Omron Sysmac Studio project Meca500_V9_1_5_Omron_EtherCat_Square_Demo_V1 (Sysmac Studio 1.47.0.64008, StandardProject)

# Controller NX1P2_9024DT1: NX1P2-9024DT1 version 1.16
Units and slaves: Node1 : Meca500 (E001)
Task PrimaryTask (priority 4, period or condition 2000): Meca500_IOs, Meca500_Sequence, Meca500_Instructions

TYPE RobotControl : STRUCT
    Deactivate : BOOL;  (* offset 0.0 *)
    Activate : BOOL;  (* offset 0.1 *)
    Home : BOOL;  (* offset 0.2 *)
    ResetError : BOOL;  (* offset 0.3 *)
    EnableSimulation : BOOL;  (* offset 0.4 *)
    EnableRecoveryMode : BOOL;  (* offset 0.5 *)
END_STRUCT END_TYPE
TYPE Meca500 : STRUCT
    Outputs : Outputs;
    Inputs : Inputs;
    CommandsID : Meca500Cmd;
END_STRUCT END_TYPE
TYPE Inputs : STRUCT
    Status : Status;  (* offset 0.0 *)
    Motion : Motion;  (* offset 4.0 *)
    Joint_Set : Joint_Set;  (* offset 16.0 *)
    EndEffector_Pose : EndEffector_Pose;  (* offset 40.0 *)
    Configurations : Configurations;  (* offset 64.0 *)
    WRF : WRF;  (* offset 68.0 *)
    TRF : TRF;  (* offset 92.0 *)
    TimeStamp : TimeStamp;  (* offset 116.0 *)
    Reserved1 : SINT;  (* offset 128.0 *)
    Reserved2 : SINT;  (* offset 132.0 *)
    Reserved3 : SINT;  (* offset 136.0 *)
    DynamicData0 : DynamicData;  (* offset 140.0 *)
    DynamicData1 : DynamicData;  (* offset 168.0 *)
    DynamicData2 : DynamicData;  (* offset 196.0 *)
    DynamicData3 : DynamicData;  (* offset 224.0 *)
END_STRUCT END_TYPE
TYPE Status : STRUCT
    Busy : BOOL;
    Activated : BOOL;
    Homed : BOOL;
    SimActivated : BOOL;
    BrakesEngaged : BOOL;
    RecoveryMode : BOOL;
    Error : UINT;
END_STRUCT END_TYPE
TYPE Motion : STRUCT
    CheckPoint : UDINT;  (* offset 0.0 *)
    MoveID : UINT;  (* offset 4.0 *)
    FifoSpace : UINT;  (* offset 6.0 *)
    Paused : BOOL;  (* offset 8.0 *)
    EOB : BOOL;  (* offset 8.1 *)
    EOM : BOOL;  (* offset 8.2 *)
    FifoCleared : BOOL;  (* offset 8.3 *)
    PStop : BOOL;  (* offset 8.4 *)
    ExcessiveTorque : BOOL;  (* offset 8.5 *)
    OfflineProgramID : UINT;  (* offset 10.0 *)
END_STRUCT END_TYPE
TYPE Joint_Set : STRUCT
    SubIndex001 : REAL;
    SubIndex002 : REAL;
    SubIndex003 : REAL;
    SubIndex004 : REAL;
    SubIndex005 : REAL;
    SubIndex006 : REAL;
END_STRUCT END_TYPE
TYPE EndEffector_Pose : STRUCT
    SubIndex001 : REAL;
    SubIndex002 : REAL;
    SubIndex003 : REAL;
    SubIndex004 : REAL;
    SubIndex005 : REAL;
    SubIndex006 : REAL;
END_STRUCT END_TYPE
TYPE Configurations : STRUCT
    Shoulder : SINT;  (* offset 0.0 *)
    Elbow : SINT;  (* offset 1.0 *)
    Wrist : SINT;  (* offset 2.0 *)
    Turn : SINT;  (* offset 3.0 *)
END_STRUCT END_TYPE
TYPE WRF : STRUCT
    SubIndex001 : REAL;
    SubIndex002 : REAL;
    SubIndex003 : REAL;
    SubIndex004 : REAL;
    SubIndex005 : REAL;
    SubIndex006 : REAL;
END_STRUCT END_TYPE
TYPE TRF : STRUCT
    SubIndex001 : REAL;
    SubIndex002 : REAL;
    SubIndex003 : REAL;
    SubIndex004 : REAL;
    SubIndex005 : REAL;
    SubIndex006 : REAL;
END_STRUCT END_TYPE
TYPE TimeStamp : STRUCT
    Seconds : UDINT;
    MicroSeconds : UDINT;
    DynamicDataCycles : UDINT;
END_STRUCT END_TYPE
TYPE DynamicData : STRUCT
    DynamicDataType : UDINT;
    DynamicDataValue0 : REAL;
    DynamicDataValue1 : REAL;
    DynamicDataValue2 : REAL;
    DynamicDataValue3 : REAL;
    DynamicDataValue4 : REAL;
    DynamicDataValue5 : REAL;
END_STRUCT END_TYPE
TYPE Outputs : STRUCT
    RobotControl : RobotControl;  (* offset 0.0 *)
    MotionControl : MotionControl;  (* offset 4.0 *)
    MotionCommand : MotionCommand;  (* offset 8.0 *)
    HostTime : UDINT;  (* offset 36.0 *)
    BrakesControlAllowed : BOOL;  (* offset 40.0 *)
    BrakesEngaged : BOOL;  (* offset 40.1 *)
    DynamicDataCfg0 : UDINT;  (* offset 42.0 *)
    DynamicDataCfg1 : UDINT;  (* offset 46.0 *)
    DynamicDataCfg2 : UDINT;  (* offset 50.0 *)
    DynamicDataCfg3 : UDINT;  (* offset 56.0 *)
END_STRUCT END_TYPE
TYPE MotionControl : STRUCT
    MoveID : UINT;  (* offset 0.0 *)
    Setpoint : BOOL;  (* offset 2.0 *)
    Pause : BOOL;  (* offset 2.1 *)
    CleaMove : BOOL;  (* offset 2.2 *)
    ResetPStop2 : BOOL;  (* offset 2.3 *)
END_STRUCT END_TYPE
TYPE MotionCommand : STRUCT
    MoveCommand : UDINT;  (* offset 0.0 *)
    MoveSubIndex001 : REAL;  (* offset 4.0 *)
    MoveSubIndex002 : REAL;  (* offset 8.0 *)
    MoveSubIndex003 : REAL;  (* offset 12.0 *)
    MoveSubIndex004 : REAL;  (* offset 16.0 *)
    MoveSubIndex005 : REAL;  (* offset 20.0 *)
    MoveSubIndex006 : REAL;  (* offset 24.0 *)
END_STRUCT END_TYPE
TYPE Meca500Cmd : (NoCmd := 0, MoveJoints := 1, MovePose := 2, MoveLin := 3, MoveLinRelTrf := 4, MoveLinRelWrf := 5, Delay := 6, SetBlending := 7, SetJointVel := 8, SetJointAcc := 9, SetCartAngVel := 10, SetCartLinVel := 11, SetCartAcc := 12, SetTrf := 13, SetWrf := 14, SetConf := 15, SetAutoConf := 16, SetCheckpoint := 17, Gripper := 18, SetGripperVel := 19, SetGripperForce := 20, MoveJointsVel := 21, MoveLinVelWrf := 22, MoveLinVelTrf := 23, SetVelTimeout := 24, SetConfTurn := 25, SetAutoConfTurn := 26, SetTorqueLimits := 27, SetTorquesLimitCfg := 28, MoveJointsRel := 29, SetValveState := 30, SetGripperRange := 31, MoveGripper := 32, StartProgram := 100); END_TYPE

VAR_GLOBAL
    E001 : Meca500;  (* Robot Structure *)
    Position : ARRAY[0..5] OF real;  (* Array for positions *)
    StepSquareMove : INT;  (* Sequencer step *)
    MoveJoint1Buffered : BOOL;
    MovePose1Buffered : BOOL;
    MoveLin1Buffered : BOOL;
    SetCartLinVel1Buffered : BOOL;
    E001_Robot_Control_Deactivate_7200_01 : BOOL;  (* at ECAT://node#1/Robot Control_Deactivate_7200_01 *)
    E001_Robot_Control_Activate_7200_02 : BOOL;  (* at ECAT://node#1/Robot Control_Activate_7200_02 *)
    E001_Robot_Control_Home_7200_03 : BOOL;  (* at ECAT://node#1/Robot Control_Home_7200_03 *)
    E001_Robot_Control_Reset_Error_7200_04 : BOOL;  (* at ECAT://node#1/Robot Control_Reset Error_7200_04 *)
    E001_Robot_Control_Sim_Mode_7200_05 : BOOL;  (* at ECAT://node#1/Robot Control_Sim Mode_7200_05 *)
    E001_Robot_Control_Recovery_Mode_7200_06 : BOOL;  (* at ECAT://node#1/Robot Control_Recovery Mode_7200_06 *)
    E001_Motion_Control_Move_ID_7310_01 : UINT;  (* at ECAT://node#1/Motion Control_Move ID_7310_01 *)
    E001_Motion_Control_SetPoint_7310_02 : BOOL;  (* at ECAT://node#1/Motion Control_SetPoint_7310_02 *)
    E001_Motion_Control_Pause_7310_03 : BOOL;  (* at ECAT://node#1/Motion Control_Pause_7310_03 *)
    E001_Motion_Control_Clear_Move_7310_04 : BOOL;  (* at ECAT://node#1/Motion Control_Clear Move_7310_04 *)
    E001_Motion_Control_Reset_PStop2_7310_05 : BOOL;  (* at ECAT://node#1/Motion Control_Reset PStop2_7310_05 *)
    E001_Move_Move_Command_7305_00 : UDINT;  (* at ECAT://node#1/Move_Move Command_7305_00 *)
    E001_Move_SubIndex_001_7306_01 : REAL;  (* at ECAT://node#1/Move_SubIndex 001_7306_01 *)
    E001_Move_SubIndex_002_7306_02 : REAL;  (* at ECAT://node#1/Move_SubIndex 002_7306_02 *)
    E001_Move_SubIndex_003_7306_03 : REAL;  (* at ECAT://node#1/Move_SubIndex 003_7306_03 *)
    E001_Move_SubIndex_004_7306_04 : REAL;  (* at ECAT://node#1/Move_SubIndex 004_7306_04 *)
    E001_Move_SubIndex_005_7306_05 : REAL;  (* at ECAT://node#1/Move_SubIndex 005_7306_05 *)
    E001_Move_SubIndex_006_7306_06 : REAL;  (* at ECAT://node#1/Move_SubIndex 006_7306_06 *)
    E001_Host_Time_Host_Time_7400_00 : UDINT;  (* at ECAT://node#1/Host Time_Host Time_7400_00 *)
    E001_Brakes_Control_BrakesControlAllowed_7410_01 : BOOL;  (* at ECAT://node#1/Brakes Control_BrakesControlAllowed_7410_01 *)
    E001_Brakes_Control_BrakesEngaged_7410_02 : BOOL;  (* at ECAT://node#1/Brakes Control_BrakesEngaged_7410_02 *)
    E001_Dynamic_Data_Cfg_0_Dynamic_Type_7420_01 : UDINT;  (* at ECAT://node#1/Dynamic Data Cfg 0_Dynamic Type_7420_01 *)
    E001_Dynamic_Data_Cfg_1_Dynamic_Type_7421_01 : UDINT;  (* at ECAT://node#1/Dynamic Data Cfg 1_Dynamic Type_7421_01 *)
    E001_Dynamic_Data_Cfg_2_Dynamic_Type_7422_01 : UDINT;  (* at ECAT://node#1/Dynamic Data Cfg 2_Dynamic Type_7422_01 *)
    E001_Dynamic_Data_Cfg_3_Dynamic_Type_7423_01 : UDINT;  (* at ECAT://node#1/Dynamic Data Cfg 3_Dynamic Type_7423_01 *)
    E001_Robot_Status_Busy_6010_02 : BOOL;  (* at ECAT://node#1/Robot Status_Busy_6010_02 *)
    E001_Robot_Status_Activated_6010_03 : BOOL;  (* at ECAT://node#1/Robot Status_Activated_6010_03 *)
    E001_Robot_Status_Homed_6010_04 : BOOL;  (* at ECAT://node#1/Robot Status_Homed_6010_04 *)
    E001_Robot_Status_SimActivated_6010_05 : BOOL;  (* at ECAT://node#1/Robot Status_SimActivated_6010_05 *)
    E001_Robot_Status_BrakesEngaged_6010_06 : BOOL;  (* at ECAT://node#1/Robot Status_BrakesEngaged_6010_06 *)
    E001_Robot_Status_RecoveryMode_6010_07 : BOOL;  (* at ECAT://node#1/Robot Status_RecoveryMode_6010_07 *)
    E001_Robot_Status_Error_6010_01 : UINT;  (* at ECAT://node#1/Robot Status_Error_6010_01 *)
    E001_Motion_Status_CheckPoint_6015_01 : UDINT;  (* at ECAT://node#1/Motion Status_CheckPoint_6015_01 *)
    E001_Motion_Status_Move_ID_6015_02 : UINT;  (* at ECAT://node#1/Motion Status_Move ID_6015_02 *)
    E001_Motion_Status_FIFO_Space_6015_03 : UINT;  (* at ECAT://node#1/Motion Status_FIFO Space_6015_03 *)
    E001_Motion_Status_Paused_6015_05 : BOOL;  (* at ECAT://node#1/Motion Status_Paused_6015_05 *)
    E001_Motion_Status_EOB_6015_06 : BOOL;  (* at ECAT://node#1/Motion Status_EOB_6015_06 *)
    E001_Motion_Status_EOM_6015_07 : BOOL;  (* at ECAT://node#1/Motion Status_EOM_6015_07 *)
    E001_Motion_Status_FIFO_Cleared_6015_08 : BOOL;  (* at ECAT://node#1/Motion Status_FIFO Cleared_6015_08 *)
    E001_Motion_Status_PStop2_6015_09 : BOOL;  (* at ECAT://node#1/Motion Status_PStop2_6015_09 *)
    E001_Motion_Status_Excessive_torque_6015_0A : BOOL;  (* at ECAT://node#1/Motion Status_Excessive torque_6015_0A *)
    E001_Motion_Status_Offline_Program_ID_6015_04 : UINT;  (* at ECAT://node#1/Motion Status_Offline Program ID_6015_04 *)
    E001_Joint_Set_SubIndex_001_6030_01 : REAL;  (* at ECAT://node#1/Joint Set_SubIndex 001_6030_01 *)
    E001_Joint_Set_SubIndex_002_6030_02 : REAL;  (* at ECAT://node#1/Joint Set_SubIndex 002_6030_02 *)
    E001_Joint_Set_SubIndex_003_6030_03 : REAL;  (* at ECAT://node#1/Joint Set_SubIndex 003_6030_03 *)
    E001_Joint_Set_SubIndex_004_6030_04 : REAL;  (* at ECAT://node#1/Joint Set_SubIndex 004_6030_04 *)
    E001_Joint_Set_SubIndex_005_6030_05 : REAL;  (* at ECAT://node#1/Joint Set_SubIndex 005_6030_05 *)
    E001_Joint_Set_SubIndex_006_6030_06 : REAL;  (* at ECAT://node#1/Joint Set_SubIndex 006_6030_06 *)
    E001_End_Effector_Pose_SubIndex_001_6031_01 : REAL;  (* at ECAT://node#1/End-Effector Pose_SubIndex 001_6031_01 *)
    E001_End_Effector_Pose_SubIndex_002_6031_02 : REAL;  (* at ECAT://node#1/End-Effector Pose_SubIndex 002_6031_02 *)
    E001_End_Effector_Pose_SubIndex_003_6031_03 : REAL;  (* at ECAT://node#1/End-Effector Pose_SubIndex 003_6031_03 *)
    E001_End_Effector_Pose_SubIndex_004_6031_04 : REAL;  (* at ECAT://node#1/End-Effector Pose_SubIndex 004_6031_04 *)
    E001_End_Effector_Pose_SubIndex_005_6031_05 : REAL;  (* at ECAT://node#1/End-Effector Pose_SubIndex 005_6031_05 *)
    E001_End_Effector_Pose_SubIndex_006_6031_06 : REAL;  (* at ECAT://node#1/End-Effector Pose_SubIndex 006_6031_06 *)
    E001_Configurations_Shoulder_6046_01 : SINT;  (* at ECAT://node#1/Configurations_Shoulder_6046_01 *)
    E001_Configurations_Elbow_6046_02 : SINT;  (* at ECAT://node#1/Configurations_Elbow_6046_02 *)
    E001_Configurations_Wrist_6046_03 : SINT;  (* at ECAT://node#1/Configurations_Wrist_6046_03 *)
    E001_Configurations_Turn_6046_04 : SINT;  (* at ECAT://node#1/Configurations_Turn_6046_04 *)
    E001_WRF_SubIndex_001_6050_01 : REAL;  (* at ECAT://node#1/WRF_SubIndex 001_6050_01 *)
    E001_WRF_SubIndex_002_6050_02 : REAL;  (* at ECAT://node#1/WRF_SubIndex 002_6050_02 *)
    E001_WRF_SubIndex_003_6050_03 : REAL;  (* at ECAT://node#1/WRF_SubIndex 003_6050_03 *)
    E001_WRF_SubIndex_004_6050_04 : REAL;  (* at ECAT://node#1/WRF_SubIndex 004_6050_04 *)
    E001_WRF_SubIndex_005_6050_05 : REAL;  (* at ECAT://node#1/WRF_SubIndex 005_6050_05 *)
    E001_WRF_SubIndex_006_6050_06 : REAL;  (* at ECAT://node#1/WRF_SubIndex 006_6050_06 *)
    E001_TRF_SubIndex_001_6051_01 : REAL;  (* at ECAT://node#1/TRF_SubIndex 001_6051_01 *)
    E001_TRF_SubIndex_002_6051_02 : REAL;  (* at ECAT://node#1/TRF_SubIndex 002_6051_02 *)
    E001_TRF_SubIndex_003_6051_03 : REAL;  (* at ECAT://node#1/TRF_SubIndex 003_6051_03 *)
    E001_TRF_SubIndex_004_6051_04 : REAL;  (* at ECAT://node#1/TRF_SubIndex 004_6051_04 *)
    E001_TRF_SubIndex_005_6051_05 : REAL;  (* at ECAT://node#1/TRF_SubIndex 005_6051_05 *)
    E001_TRF_SubIndex_006_6051_06 : REAL;  (* at ECAT://node#1/TRF_SubIndex 006_6051_06 *)
    E001_Robot_Timestamp_Timestamp_Seconds_6060_01 : UDINT;  (* at ECAT://node#1/Robot Timestamp_Timestamp Seconds_6060_01 *)
    E001_Robot_Timestamp_Timestamp_Microseconds_6060_02 : UDINT;  (* at ECAT://node#1/Robot Timestamp_Timestamp Microseconds_6060_02 *)
    E001_Robot_Timestamp_Dynamic_Data_Cycles_6060_03 : UDINT;  (* at ECAT://node#1/Robot Timestamp_Dynamic Data Cycles_6060_03 *)
    E001_Dynamic_Data_0_Dynamic_Type_6070_01 : UDINT;  (* at ECAT://node#1/Dynamic Data 0_Dynamic Type_6070_01 *)
    E001_Dynamic_Data_0_Value_0_6070_02 : REAL;  (* at ECAT://node#1/Dynamic Data 0_Value 0_6070_02 *)
    E001_Dynamic_Data_0_Value_1_6070_03 : REAL;  (* at ECAT://node#1/Dynamic Data 0_Value 1_6070_03 *)
    E001_Dynamic_Data_0_Value_2_6070_04 : REAL;  (* at ECAT://node#1/Dynamic Data 0_Value 2_6070_04 *)
    E001_Dynamic_Data_0_Value_3_6070_05 : REAL;  (* at ECAT://node#1/Dynamic Data 0_Value 3_6070_05 *)
    E001_Dynamic_Data_0_Value_4_6070_06 : REAL;  (* at ECAT://node#1/Dynamic Data 0_Value 4_6070_06 *)
    E001_Dynamic_Data_0_Value_5_6070_07 : REAL;  (* at ECAT://node#1/Dynamic Data 0_Value 5_6070_07 *)
    E001_Dynamic_Data_1_Dynamic_Type_6071_01 : UDINT;  (* at ECAT://node#1/Dynamic Data 1_Dynamic Type_6071_01 *)
    E001_Dynamic_Data_1_Value_0_6071_02 : REAL;  (* at ECAT://node#1/Dynamic Data 1_Value 0_6071_02 *)
    E001_Dynamic_Data_1_Value_1_6071_03 : REAL;  (* at ECAT://node#1/Dynamic Data 1_Value 1_6071_03 *)
    E001_Dynamic_Data_1_Value_2_6071_04 : REAL;  (* at ECAT://node#1/Dynamic Data 1_Value 2_6071_04 *)
    E001_Dynamic_Data_1_Value_3_6071_05 : REAL;  (* at ECAT://node#1/Dynamic Data 1_Value 3_6071_05 *)
    E001_Dynamic_Data_1_Value_4_6071_06 : REAL;  (* at ECAT://node#1/Dynamic Data 1_Value 4_6071_06 *)
    E001_Dynamic_Data_1_Value_5_6071_07 : REAL;  (* at ECAT://node#1/Dynamic Data 1_Value 5_6071_07 *)
    E001_Dynamic_Data_2_Dynamic_Type_6072_01 : UDINT;  (* at ECAT://node#1/Dynamic Data 2_Dynamic Type_6072_01 *)
    E001_Dynamic_Data_2_Value_0_6072_02 : REAL;  (* at ECAT://node#1/Dynamic Data 2_Value 0_6072_02 *)
    E001_Dynamic_Data_2_Value_1_6072_03 : REAL;  (* at ECAT://node#1/Dynamic Data 2_Value 1_6072_03 *)
    E001_Dynamic_Data_2_Value_2_6072_04 : REAL;  (* at ECAT://node#1/Dynamic Data 2_Value 2_6072_04 *)
    E001_Dynamic_Data_2_Value_3_6072_05 : REAL;  (* at ECAT://node#1/Dynamic Data 2_Value 3_6072_05 *)
    E001_Dynamic_Data_2_Value_4_6072_06 : REAL;  (* at ECAT://node#1/Dynamic Data 2_Value 4_6072_06 *)
    E001_Dynamic_Data_2_Value_5_6072_07 : REAL;  (* at ECAT://node#1/Dynamic Data 2_Value 5_6072_07 *)
    E001_Dynamic_Data_3_Dynamic_Type_6073_01 : UDINT;  (* at ECAT://node#1/Dynamic Data 3_Dynamic Type_6073_01 *)
    E001_Dynamic_Data_3_Value_0_6073_02 : REAL;  (* at ECAT://node#1/Dynamic Data 3_Value 0_6073_02 *)
    E001_Dynamic_Data_3_Value_1_6073_03 : REAL;  (* at ECAT://node#1/Dynamic Data 3_Value 1_6073_03 *)
    E001_Dynamic_Data_3_Value_2_6073_04 : REAL;  (* at ECAT://node#1/Dynamic Data 3_Value 2_6073_04 *)
    E001_Dynamic_Data_3_Value_3_6073_05 : REAL;  (* at ECAT://node#1/Dynamic Data 3_Value 3_6073_05 *)
    E001_Dynamic_Data_3_Value_4_6073_06 : REAL;  (* at ECAT://node#1/Dynamic Data 3_Value 4_6073_06 *)
    E001_Dynamic_Data_3_Value_5_6073_07 : REAL;  (* at ECAT://node#1/Dynamic Data 3_Value 5_6073_07 *)
END_VAR

PROGRAM Meca500_IOs
VAR_EXTERNAL
    E001_Robot_Control_Deactivate_7200_01 : BOOL;
    E001_Robot_Control_Activate_7200_02 : BOOL;
    E001_Robot_Control_Home_7200_03 : BOOL;
    E001_Robot_Control_Reset_Error_7200_04 : BOOL;
    E001_Robot_Control_Sim_Mode_7200_05 : BOOL;
    E001_Robot_Control_Recovery_Mode_7200_06 : BOOL;
    E001_Motion_Control_Move_ID_7310_01 : UINT;
    E001_Motion_Control_SetPoint_7310_02 : BOOL;
    E001_Motion_Control_Pause_7310_03 : BOOL;
    E001_Motion_Control_Clear_Move_7310_04 : BOOL;
    E001_Motion_Control_Reset_PStop2_7310_05 : BOOL;
    E001_Move_Move_Command_7305_00 : UDINT;
    E001_Move_SubIndex_001_7306_01 : REAL;
    E001_Move_SubIndex_002_7306_02 : REAL;
    E001_Move_SubIndex_003_7306_03 : REAL;
    E001_Move_SubIndex_004_7306_04 : REAL;
    E001_Move_SubIndex_005_7306_05 : REAL;
    E001_Move_SubIndex_006_7306_06 : REAL;
    E001_Host_Time_Host_Time_7400_00 : UDINT;
    E001_Brakes_Control_BrakesControlAllowed_7410_01 : BOOL;
    E001_Brakes_Control_BrakesEngaged_7410_02 : BOOL;
    E001_Dynamic_Data_Cfg_0_Dynamic_Type_7420_01 : UDINT;
    E001_Dynamic_Data_Cfg_1_Dynamic_Type_7421_01 : UDINT;
    E001_Dynamic_Data_Cfg_2_Dynamic_Type_7422_01 : UDINT;
    E001_Dynamic_Data_Cfg_3_Dynamic_Type_7423_01 : UDINT;
    E001 : Meca500;
    E001_Robot_Status_Busy_6010_02 : BOOL;
    E001_Robot_Status_Activated_6010_03 : BOOL;
    E001_Robot_Status_Homed_6010_04 : BOOL;
    E001_Robot_Status_SimActivated_6010_05 : BOOL;
    E001_Robot_Status_BrakesEngaged_6010_06 : BOOL;
    E001_Robot_Status_RecoveryMode_6010_07 : BOOL;
    E001_Robot_Status_Error_6010_01 : UINT;
    E001_Motion_Status_CheckPoint_6015_01 : UDINT;
    E001_Motion_Status_Move_ID_6015_02 : UINT;
    E001_Motion_Status_FIFO_Space_6015_03 : UINT;
    E001_Motion_Status_Paused_6015_05 : BOOL;
    E001_Motion_Status_EOB_6015_06 : BOOL;
    E001_Motion_Status_EOM_6015_07 : BOOL;
    E001_Motion_Status_FIFO_Cleared_6015_08 : BOOL;
    E001_Motion_Status_PStop2_6015_09 : BOOL;
    E001_Motion_Status_Excessive_torque_6015_0A : BOOL;
    E001_Motion_Status_Offline_Program_ID_6015_04 : UINT;
    E001_Joint_Set_SubIndex_001_6030_01 : REAL;
    E001_Joint_Set_SubIndex_002_6030_02 : REAL;
    E001_Joint_Set_SubIndex_003_6030_03 : REAL;
    E001_Joint_Set_SubIndex_004_6030_04 : REAL;
    E001_Joint_Set_SubIndex_005_6030_05 : REAL;
    E001_Joint_Set_SubIndex_006_6030_06 : REAL;
    E001_End_Effector_Pose_SubIndex_001_6031_01 : REAL;
    E001_End_Effector_Pose_SubIndex_002_6031_02 : REAL;
    E001_End_Effector_Pose_SubIndex_003_6031_03 : REAL;
    E001_End_Effector_Pose_SubIndex_004_6031_04 : REAL;
    E001_End_Effector_Pose_SubIndex_005_6031_05 : REAL;
    E001_End_Effector_Pose_SubIndex_006_6031_06 : REAL;
    E001_Configurations_Shoulder_6046_01 : SINT;
    E001_Configurations_Elbow_6046_02 : SINT;
    E001_Configurations_Wrist_6046_03 : SINT;
    E001_Configurations_Turn_6046_04 : SINT;
    E001_WRF_SubIndex_001_6050_01 : REAL;
    E001_WRF_SubIndex_002_6050_02 : REAL;
    E001_WRF_SubIndex_003_6050_03 : REAL;
    E001_WRF_SubIndex_004_6050_04 : REAL;
    E001_WRF_SubIndex_005_6050_05 : REAL;
    E001_WRF_SubIndex_006_6050_06 : REAL;
    E001_TRF_SubIndex_001_6051_01 : REAL;
    E001_TRF_SubIndex_002_6051_02 : REAL;
    E001_TRF_SubIndex_003_6051_03 : REAL;
    E001_TRF_SubIndex_004_6051_04 : REAL;
    E001_TRF_SubIndex_005_6051_05 : REAL;
    E001_TRF_SubIndex_006_6051_06 : REAL;
    E001_Robot_Timestamp_Timestamp_Seconds_6060_01 : UDINT;
    E001_Robot_Timestamp_Timestamp_Microseconds_6060_02 : UDINT;
    E001_Robot_Timestamp_Dynamic_Data_Cycles_6060_03 : UDINT;
    E001_Dynamic_Data_0_Dynamic_Type_6070_01 : UDINT;
    E001_Dynamic_Data_0_Value_0_6070_02 : REAL;
    E001_Dynamic_Data_0_Value_1_6070_03 : REAL;
    E001_Dynamic_Data_0_Value_2_6070_04 : REAL;
    E001_Dynamic_Data_0_Value_3_6070_05 : REAL;
    E001_Dynamic_Data_0_Value_4_6070_06 : REAL;
    E001_Dynamic_Data_0_Value_5_6070_07 : REAL;
    E001_Dynamic_Data_1_Dynamic_Type_6071_01 : UDINT;
    E001_Dynamic_Data_1_Value_0_6071_02 : REAL;
    E001_Dynamic_Data_1_Value_1_6071_03 : REAL;
    E001_Dynamic_Data_1_Value_2_6071_04 : REAL;
    E001_Dynamic_Data_1_Value_3_6071_05 : REAL;
    E001_Dynamic_Data_1_Value_4_6071_06 : REAL;
    E001_Dynamic_Data_1_Value_5_6071_07 : REAL;
    E001_Dynamic_Data_2_Dynamic_Type_6072_01 : UDINT;
    E001_Dynamic_Data_2_Value_0_6072_02 : REAL;
    E001_Dynamic_Data_2_Value_1_6072_03 : REAL;
    E001_Dynamic_Data_2_Value_2_6072_04 : REAL;
    E001_Dynamic_Data_2_Value_3_6072_05 : REAL;
    E001_Dynamic_Data_2_Value_4_6072_06 : REAL;
    E001_Dynamic_Data_2_Value_5_6072_07 : REAL;
    E001_Dynamic_Data_3_Dynamic_Type_6073_01 : UDINT;
    E001_Dynamic_Data_3_Value_0_6073_02 : REAL;
    E001_Dynamic_Data_3_Value_1_6073_03 : REAL;
    E001_Dynamic_Data_3_Value_2_6073_04 : REAL;
    E001_Dynamic_Data_3_Value_3_6073_05 : REAL;
    E001_Dynamic_Data_3_Value_4_6073_06 : REAL;
    E001_Dynamic_Data_3_Value_5_6073_07 : REAL;
END_VAR
//Outputs
//Outputs.RobotControl
E001_Robot_Control_Deactivate_7200_01						:=	E001.Outputs.RobotControl.Deactivate;
E001_Robot_Control_Activate_7200_02		 					:=	E001.Outputs.RobotControl.Activate;
E001_Robot_Control_Home_7200_03		 						:=	E001.Outputs.RobotControl.Home;
E001_Robot_Control_Reset_Error_7200_04		 				:=	E001.Outputs.RobotControl.ResetError;
E001_Robot_Control_Sim_Mode_7200_05		 				:=	E001.Outputs.RobotControl.EnableSimulation;
E001_Robot_Control_Recovery_Mode_7200_06		 		:=	E001.Outputs.RobotControl.EnableRecoveryMode;

//Outputs.MotionControl
E001_Motion_Control_Move_ID_7310_01		 				:=	E001.Outputs.MotionControl.MoveID;
E001_Motion_Control_SetPoint_7310_02		 				:=	E001.Outputs.MotionControl.Setpoint;
E001_Motion_Control_Pause_7310_03		 					:=	E001.Outputs.MotionControl.Pause;
E001_Motion_Control_Clear_Move_7310_04		 			:=	E001.Outputs.MotionControl.CleaMove;
E001_Motion_Control_Reset_PStop2_7310_05		 		:=	E001.Outputs.MotionControl.ResetPStop2;

//Outputs.MotionCommand
E001_Move_Move_Command_7305_00		 					:= E001.Outputs.MotionCommand.MoveCommand;
E001_Move_SubIndex_001_7306_01		 						:=	E001.Outputs.MotionCommand.MoveSubIndex001;
E001_Move_SubIndex_002_7306_02		 						:=	E001.Outputs.MotionCommand.MoveSubIndex002;
E001_Move_SubIndex_003_7306_03		 						:=	E001.Outputs.MotionCommand.MoveSubIndex003;
E001_Move_SubIndex_004_7306_04		 						:=	E001.Outputs.MotionCommand.MoveSubIndex004;
E001_Move_SubIndex_005_7306_05		 						:=	E001.Outputs.MotionCommand.MoveSubIndex005;
E001_Move_SubIndex_006_7306_06		 						:=	E001.Outputs.MotionCommand.MoveSubIndex006;

E001_Host_Time_Host_Time_7400_00		 						:=	E001.Outputs.HostTime;
E001_Brakes_Control_BrakesControlAllowed_7410_01	:=	E001.Outputs.BrakesControlAllowed;
E001_Brakes_Control_BrakesEngaged_7410_02				:=	E001.Outputs.BrakesEngaged;
E001_Dynamic_Data_Cfg_0_Dynamic_Type_7420_01		:=	E001.Outputs.DynamicDataCfg0;
E001_Dynamic_Data_Cfg_1_Dynamic_Type_7421_01		:=	E001.Outputs.DynamicDataCfg1;
E001_Dynamic_Data_Cfg_2_Dynamic_Type_7422_01		:=	E001.Outputs.DynamicDataCfg2;
E001_Dynamic_Data_Cfg_3_Dynamic_Type_7423_01		:=	E001.Outputs.DynamicDataCfg3;

//Inputs
//Inputs.Status
E001.Inputs.Status.Busy	:=	E001_Robot_Status_Busy_6010_02;
E001.Inputs.Status.Activated	:=	E001_Robot_Status_Activated_6010_03;
E001.Inputs.Status.Homed	:=	E001_Robot_Status_Homed_6010_04;
E001.Inputs.Status.SimActivated	:=	E001_Robot_Status_SimActivated_6010_05	;
E001.Inputs.Status.BrakesEngaged	:=	E001_Robot_Status_BrakesEngaged_6010_06	;
E001.Inputs.Status.RecoveryMode	:=	E001_Robot_Status_RecoveryMode_6010_07;
E001.Inputs.Status.Error	:=	E001_Robot_Status_Error_6010_01;

//Inputs.Motion
E001.Inputs.Motion.CheckPoint	:=	E001_Motion_Status_CheckPoint_6015_01;
E001.Inputs.Motion.MoveID	:=	E001_Motion_Status_Move_ID_6015_02;
E001.Inputs.Motion.FifoSpace	:=	E001_Motion_Status_FIFO_Space_6015_03;
E001.Inputs.Motion.Paused	:=	E001_Motion_Status_Paused_6015_05;
E001.Inputs.Motion.EOB	:=	E001_Motion_Status_EOB_6015_06;
E001.Inputs.Motion.EOM	:=	E001_Motion_Status_EOM_6015_07;
E001.Inputs.Motion.FifoCleared	:=	E001_Motion_Status_FIFO_Cleared_6015_08;
E001.Inputs.Motion.PStop	:=		E001_Motion_Status_PStop2_6015_09;
E001.Inputs.Motion.ExcessiveTorque	:=	E001_Motion_Status_Excessive_torque_6015_0A;
E001.Inputs.Motion.OfflineProgramID	:=	E001_Motion_Status_Offline_Program_ID_6015_04;

//Inputs.Joints
E001.Inputs.Joint_Set.SubIndex001	:=	E001_Joint_Set_SubIndex_001_6030_01;
E001.Inputs.Joint_Set.SubIndex002	:=	E001_Joint_Set_SubIndex_002_6030_02;
E001.Inputs.Joint_Set.SubIndex003	:=E001_Joint_Set_SubIndex_003_6030_03;
E001.Inputs.Joint_Set.SubIndex004	:=E001_Joint_Set_SubIndex_004_6030_04;
E001.Inputs.Joint_Set.SubIndex005	:=E001_Joint_Set_SubIndex_005_6030_05;
E001.Inputs.Joint_Set.SubIndex006	:=E001_Joint_Set_SubIndex_006_6030_06;

//Inputs.EndEffector
E001.Inputs.EndEffector_Pose.SubIndex001	:=	E001_End_Effector_Pose_SubIndex_001_6031_01;
E001.Inputs.EndEffector_Pose.SubIndex002	:=	E001_End_Effector_Pose_SubIndex_002_6031_02;
E001.Inputs.EndEffector_Pose.SubIndex003	:=	E001_End_Effector_Pose_SubIndex_003_6031_03;
E001.Inputs.EndEffector_Pose.SubIndex004	:=	E001_End_Effector_Pose_SubIndex_004_6031_04;
E001.Inputs.EndEffector_Pose.SubIndex005	:=	E001_End_Effector_Pose_SubIndex_005_6031_05;
E001.Inputs.EndEffector_Pose.SubIndex006	:=	E001_End_Effector_Pose_SubIndex_006_6031_06;

//Inputs.Configuration
E001.Inputs.Configurations.Shoulder	:=	E001_Configurations_Shoulder_6046_01;
E001.Inputs.Configurations.Elbow	:=	E001_Configurations_Elbow_6046_02;
E001.Inputs.Configurations.Wrist	:=	E001_Configurations_Wrist_6046_03;
E001.Inputs.Configurations.Turn	:=	E001_Configurations_Turn_6046_04;

//Inputs.WRF
E001.Inputs.WRF.SubIndex001	:=	E001_WRF_SubIndex_001_6050_01;
E001.Inputs.WRF.SubIndex002	:=	E001_WRF_SubIndex_002_6050_02;
E001.Inputs.WRF.SubIndex003	:=	E001_WRF_SubIndex_003_6050_03;
E001.Inputs.WRF.SubIndex004	:=	E001_WRF_SubIndex_004_6050_04;
E001.Inputs.WRF.SubIndex005	:=	E001_WRF_SubIndex_005_6050_05;
E001.Inputs.WRF.SubIndex006	:=	E001_WRF_SubIndex_006_6050_06;

//Inputs.TRF
E001.Inputs.TRF.SubIndex001	:=	E001_TRF_SubIndex_001_6051_01;
E001.Inputs.TRF.SubIndex002	:=	E001_TRF_SubIndex_002_6051_02;
E001.Inputs.TRF.SubIndex003	:=	E001_TRF_SubIndex_003_6051_03;
E001.Inputs.TRF.SubIndex004	:=	E001_TRF_SubIndex_004_6051_04;
E001.Inputs.TRF.SubIndex005	:=	E001_TRF_SubIndex_005_6051_05;
E001.Inputs.TRF.SubIndex006	:=	E001_TRF_SubIndex_006_6051_06;

//Inputs.TimeStamps
E001.Inputs.TimeStamp.Seconds							:=	E001_Robot_Timestamp_Timestamp_Seconds_6060_01;
E001.Inputs.TimeStamp.MicroSeconds				:=	E001_Robot_Timestamp_Timestamp_Microseconds_6060_02;
E001.Inputs.TimeStamp.DynamicDataCycles		:=	E001_Robot_Timestamp_Dynamic_Data_Cycles_6060_03;

//Inputs.DynamicData0
E001.Inputs.DynamicData0.DynamicDataType		:=	E001_Dynamic_Data_0_Dynamic_Type_6070_01;
E001.Inputs.DynamicData0.DynamicDataValue0		:=	E001_Dynamic_Data_0_Value_0_6070_02;
E001.Inputs.DynamicData0.DynamicDataValue1		:=E001_Dynamic_Data_0_Value_1_6070_03;
E001.Inputs.DynamicData0.DynamicDataValue2		:=E001_Dynamic_Data_0_Value_2_6070_04;
E001.Inputs.DynamicData0.DynamicDataValue3		:=E001_Dynamic_Data_0_Value_3_6070_05;
E001.Inputs.DynamicData0.DynamicDataValue4		:=E001_Dynamic_Data_0_Value_4_6070_06;
E001.Inputs.DynamicData0.DynamicDataValue5		:=E001_Dynamic_Data_0_Value_5_6070_07;

//Inputs.DynamicData1
E001.Inputs.DynamicData1.DynamicDataType		:=E001_Dynamic_Data_1_Dynamic_Type_6071_01;
E001.Inputs.DynamicData1.DynamicDataValue0		:=	E001_Dynamic_Data_1_Value_0_6071_02;
E001.Inputs.DynamicData1.DynamicDataValue1		:=	E001_Dynamic_Data_1_Value_1_6071_03;
E001.Inputs.DynamicData1.DynamicDataValue2		:=	E001_Dynamic_Data_1_Value_2_6071_04;
E001.Inputs.DynamicData1.DynamicDataValue3		:=	E001_Dynamic_Data_1_Value_3_6071_05;
E001.Inputs.DynamicData1.DynamicDataValue4		:=	E001_Dynamic_Data_1_Value_4_6071_06;
E001.Inputs.DynamicData1.DynamicDataValue5		:=	E001_Dynamic_Data_1_Value_5_6071_07;

//Inputs.DynamicData2
E001.Inputs.DynamicData2.DynamicDataType		:=	E001_Dynamic_Data_2_Dynamic_Type_6072_01;
E001.Inputs.DynamicData2.DynamicDataValue0		:=E001_Dynamic_Data_2_Value_0_6072_02;
E001.Inputs.DynamicData2.DynamicDataValue1		:=E001_Dynamic_Data_2_Value_1_6072_03;
E001.Inputs.DynamicData2.DynamicDataValue2		:=E001_Dynamic_Data_2_Value_2_6072_04;
E001.Inputs.DynamicData2.DynamicDataValue3		:=E001_Dynamic_Data_2_Value_3_6072_05;
E001.Inputs.DynamicData2.DynamicDataValue4		:=E001_Dynamic_Data_2_Value_4_6072_06;
E001.Inputs.DynamicData2.DynamicDataValue5		:=E001_Dynamic_Data_2_Value_5_6072_07;

//Inputs.DynamicData3
E001.Inputs.DynamicData3.DynamicDataType		:=E001_Dynamic_Data_3_Dynamic_Type_6073_01;
E001.Inputs.DynamicData3.DynamicDataValue0		:=E001_Dynamic_Data_3_Value_0_6073_02;
E001.Inputs.DynamicData3.DynamicDataValue1		:=E001_Dynamic_Data_3_Value_1_6073_03;
E001.Inputs.DynamicData3.DynamicDataValue2		:=E001_Dynamic_Data_3_Value_2_6073_04;
E001.Inputs.DynamicData3.DynamicDataValue3		:=E001_Dynamic_Data_3_Value_3_6073_05;
E001.Inputs.DynamicData3.DynamicDataValue4		:=E001_Dynamic_Data_3_Value_4_6073_06;
E001.Inputs.DynamicData3.DynamicDataValue5		:=E001_Dynamic_Data_3_Value_5_6073_07;
END_PROGRAM

PROGRAM Meca500_Sequence
VAR
    Activate : BOOL;
    Home : BOOL;
    ResetError : BOOL;
    Pause : BOOL;
    StartSequence : BOOL;  (* Start Sequence *)
END_VAR
VAR_EXTERNAL
    Position : ARRAY[0..5] OF real;
    StepSquareMove : INT;
    MoveJoint1Buffered : BOOL;
    MovePose1Buffered : BOOL;
    MoveLin1Buffered : BOOL;
    SetCartLinVel1Buffered : BOOL;
    E001 : Meca500;
END_VAR
VAR
    _e1 : R_TRIG;
END_VAR

(* Section Sequence: ladder, written here as Structured Text *)

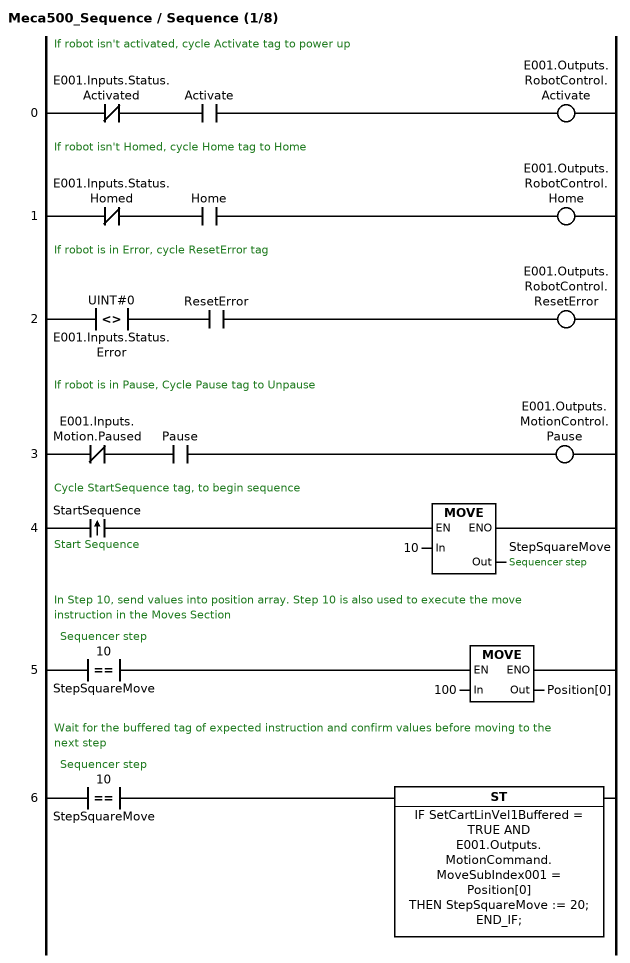
(* Rung 0: If robot isn't activated, cycle Activate tag to power up *)
E001.Outputs.RobotControl.Activate := NOT E001.Inputs.Status.Activated AND Activate;
(* Rung 1: If robot isn't Homed, cycle Home tag to Home *)
E001.Outputs.RobotControl.Home := NOT E001.Inputs.Status.Homed AND Home;
(* Rung 2: If robot is in Error, cycle ResetError tag *)
E001.Outputs.RobotControl.ResetError := (UINT#0 <> E001.Inputs.Status.Error) AND ResetError;
(* Rung 3: If robot is in Pause, Cycle Pause tag to Unpause *)
E001.Outputs.MotionControl.Pause := NOT E001.Inputs.Motion.Paused AND Pause;
(* Rung 4: Cycle StartSequence tag, to begin sequence *)
_e1(CLK := StartSequence);
IF _e1.Q THEN StepSquareMove := 10; END_IF;
(* Rung 5: In Step 10, send values into position array. Step 10 is also used to execute the move instruction in the Moves Section *)
IF 10 = StepSquareMove THEN Position[0] := 100; END_IF;
(* Rung 6: Wait for the buffered tag of expected instruction and confirm values before moving to the next step *)
IF 10 = StepSquareMove THEN
    IF SetCartLinVel1Buffered = TRUE AND
    	E001.Outputs.MotionCommand.MoveSubIndex001 = Position[0]
    	THEN StepSquareMove := 20;
    END_IF;
END_IF;

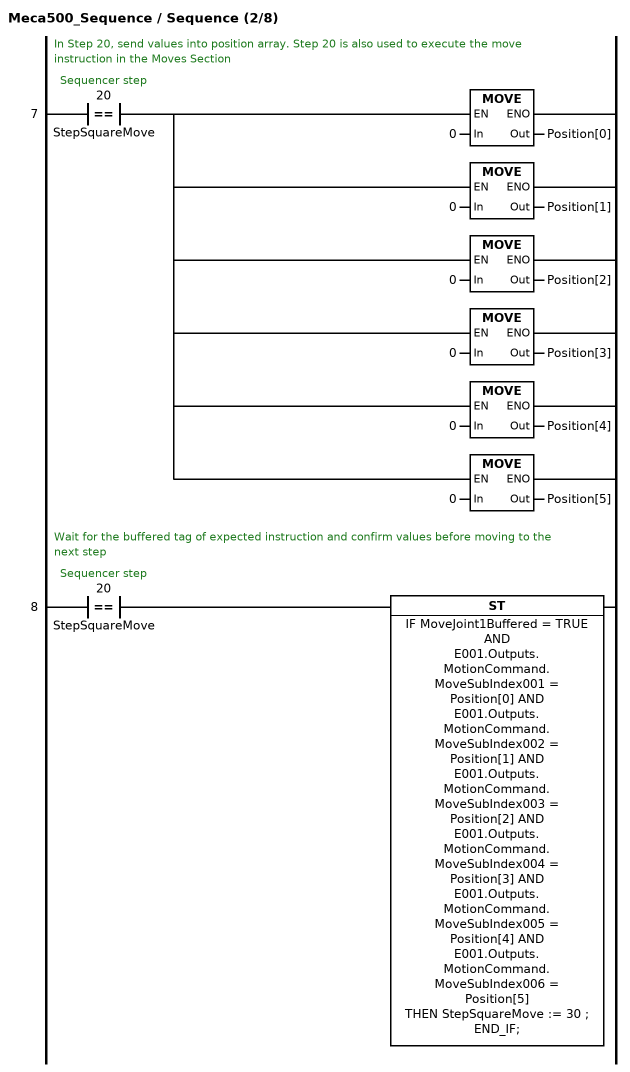
(* Rung 7: In Step 20, send values into position array. Step 20 is also used to execute the move instruction in the Moves Section *)
IF 20 = StepSquareMove THEN
    Position[0] := 0;
    Position[1] := 0;
    Position[2] := 0;
    Position[3] := 0;
    Position[4] := 0;
    Position[5] := 0;
END_IF;
(* Rung 8: Wait for the buffered tag of expected instruction and confirm values before moving to the next step *)
IF 20 = StepSquareMove THEN
    IF MoveJoint1Buffered = TRUE AND
    	E001.Outputs.MotionCommand.MoveSubIndex001 = Position[0] AND
    	E001.Outputs.MotionCommand.MoveSubIndex002 = Position[1] AND
    	E001.Outputs.MotionCommand.MoveSubIndex003 = Position[2] AND
    	E001.Outputs.MotionCommand.MoveSubIndex004 = Position[3] AND
    	E001.Outputs.MotionCommand.MoveSubIndex005 = Position[4] AND
    	E001.Outputs.MotionCommand.MoveSubIndex006 = Position[5] 
    	THEN StepSquareMove := 30 ;
    END_IF;
END_IF;

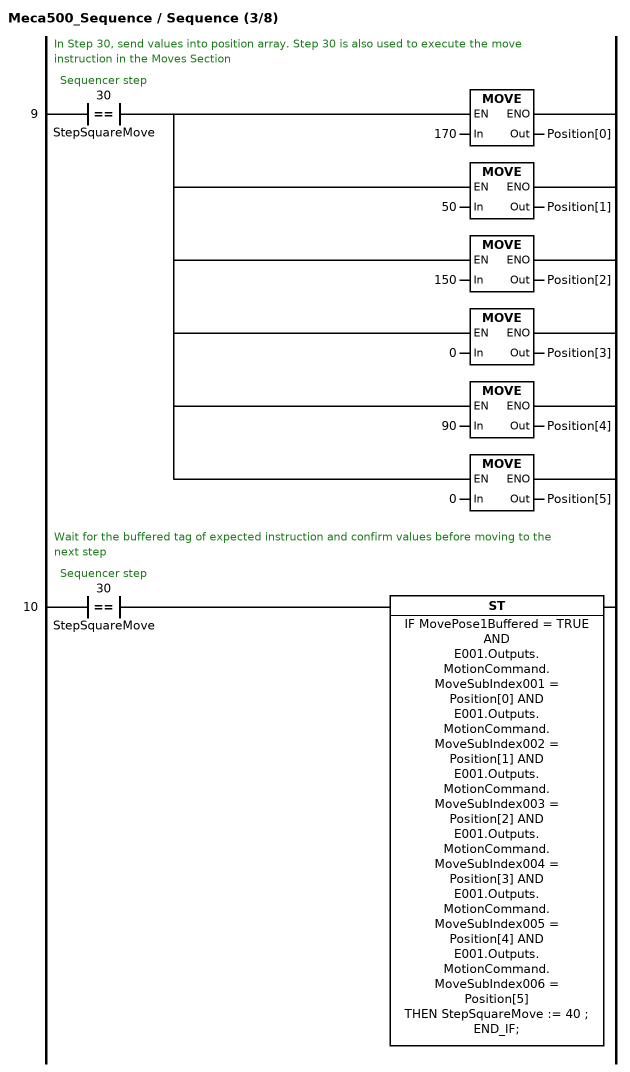
(* Rung 9: In Step 30, send values into position array. Step 30 is also used to execute the move instruction in the Moves Section *)
IF 30 = StepSquareMove THEN
    Position[0] := 170;
    Position[1] := 50;
    Position[2] := 150;
    Position[3] := 0;
    Position[4] := 90;
    Position[5] := 0;
END_IF;
(* Rung 10: Wait for the buffered tag of expected instruction and confirm values before moving to the next step *)
IF 30 = StepSquareMove THEN
    IF MovePose1Buffered = TRUE AND
    	E001.Outputs.MotionCommand.MoveSubIndex001 = Position[0] AND
    	E001.Outputs.MotionCommand.MoveSubIndex002 = Position[1] AND
    	E001.Outputs.MotionCommand.MoveSubIndex003 = Position[2] AND
    	E001.Outputs.MotionCommand.MoveSubIndex004 = Position[3] AND
    	E001.Outputs.MotionCommand.MoveSubIndex005 = Position[4] AND
    	E001.Outputs.MotionCommand.MoveSubIndex006 = Position[5] 
    	THEN StepSquareMove := 40 ;
    END_IF;
END_IF;

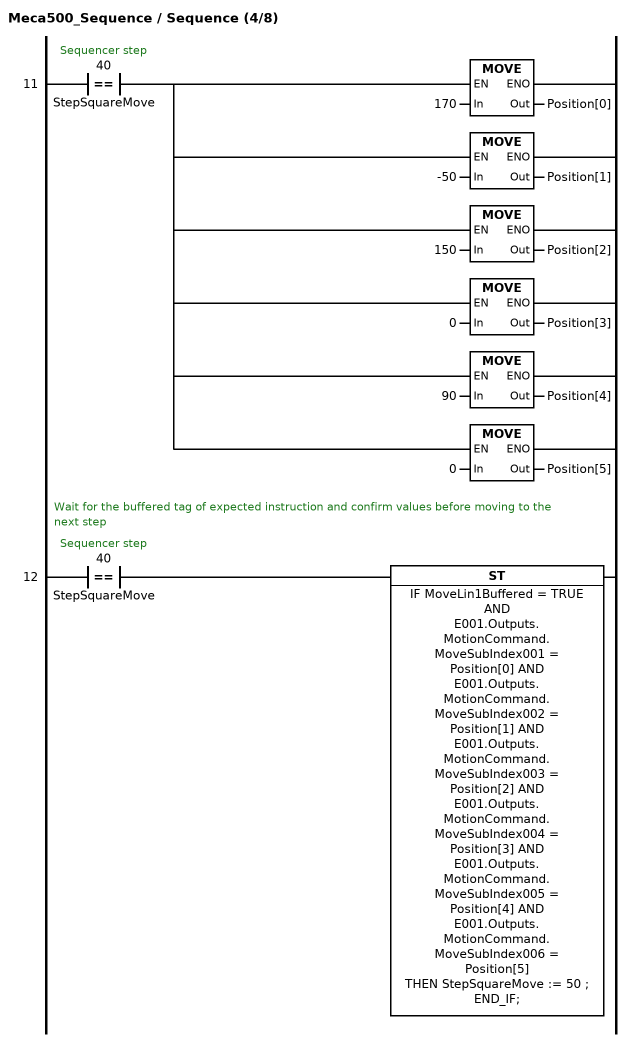
(* Rung 11 *)
IF 40 = StepSquareMove THEN
    Position[0] := 170;
    Position[1] := -50;
    Position[2] := 150;
    Position[3] := 0;
    Position[4] := 90;
    Position[5] := 0;
END_IF;
(* Rung 12: Wait for the buffered tag of expected instruction and confirm values before moving to the next step *)
IF 40 = StepSquareMove THEN
    IF MoveLin1Buffered = TRUE AND
    	E001.Outputs.MotionCommand.MoveSubIndex001 = Position[0] AND
    	E001.Outputs.MotionCommand.MoveSubIndex002 = Position[1] AND
    	E001.Outputs.MotionCommand.MoveSubIndex003 = Position[2] AND
    	E001.Outputs.MotionCommand.MoveSubIndex004 = Position[3] AND
    	E001.Outputs.MotionCommand.MoveSubIndex005 = Position[4] AND
    	E001.Outputs.MotionCommand.MoveSubIndex006 = Position[5] 
    	THEN StepSquareMove := 50 ;
    END_IF;
END_IF;

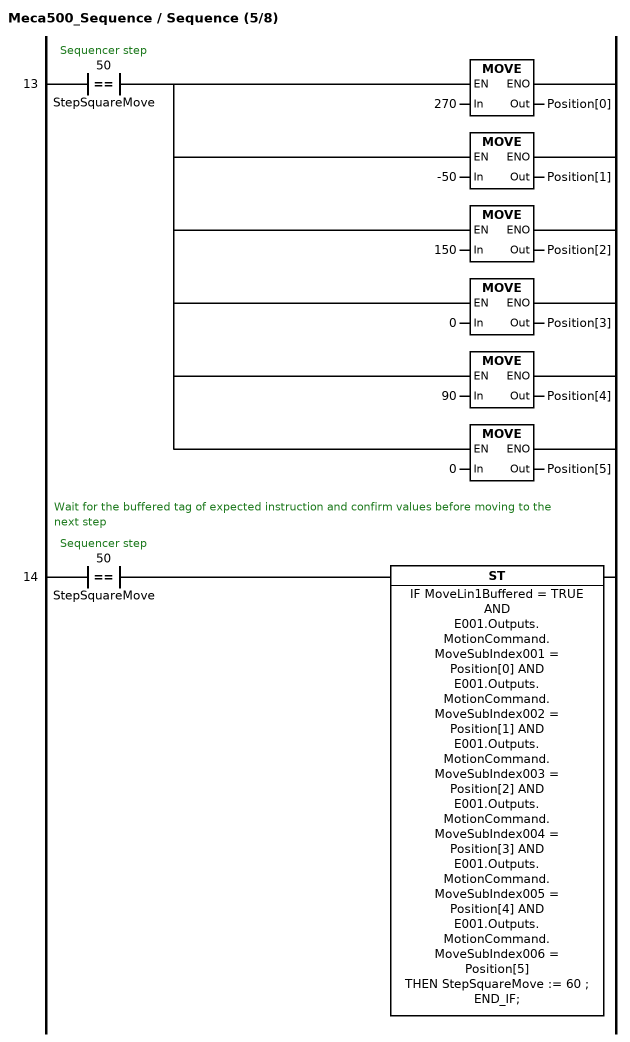
(* Rung 13 *)
IF 50 = StepSquareMove THEN
    Position[0] := 270;
    Position[1] := -50;
    Position[2] := 150;
    Position[3] := 0;
    Position[4] := 90;
    Position[5] := 0;
END_IF;
(* Rung 14: Wait for the buffered tag of expected instruction and confirm values before moving to the next step *)
IF 50 = StepSquareMove THEN
    IF MoveLin1Buffered = TRUE AND
    	E001.Outputs.MotionCommand.MoveSubIndex001 = Position[0] AND
    	E001.Outputs.MotionCommand.MoveSubIndex002 = Position[1] AND
    	E001.Outputs.MotionCommand.MoveSubIndex003 = Position[2] AND
    	E001.Outputs.MotionCommand.MoveSubIndex004 = Position[3] AND
    	E001.Outputs.MotionCommand.MoveSubIndex005 = Position[4] AND
    	E001.Outputs.MotionCommand.MoveSubIndex006 = Position[5] 
    	THEN StepSquareMove := 60 ;
    END_IF;
END_IF;

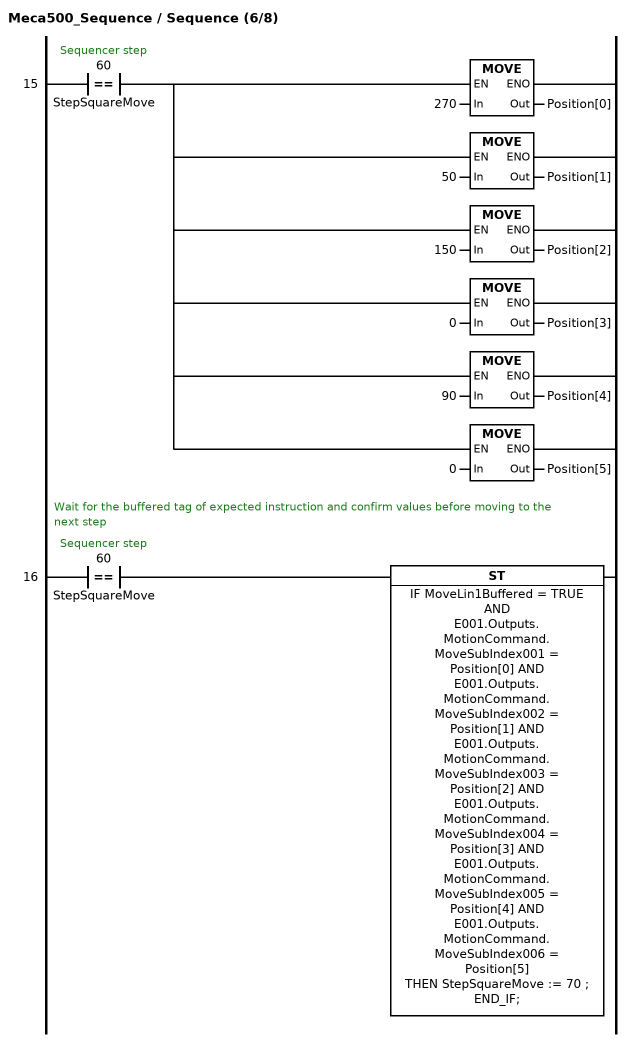
(* Rung 15 *)
IF 60 = StepSquareMove THEN
    Position[0] := 270;
    Position[1] := 50;
    Position[2] := 150;
    Position[3] := 0;
    Position[4] := 90;
    Position[5] := 0;
END_IF;
(* Rung 16: Wait for the buffered tag of expected instruction and confirm values before moving to the next step *)
IF 60 = StepSquareMove THEN
    IF MoveLin1Buffered = TRUE AND
    	E001.Outputs.MotionCommand.MoveSubIndex001 = Position[0] AND
    	E001.Outputs.MotionCommand.MoveSubIndex002 = Position[1] AND
    	E001.Outputs.MotionCommand.MoveSubIndex003 = Position[2] AND
    	E001.Outputs.MotionCommand.MoveSubIndex004 = Position[3] AND
    	E001.Outputs.MotionCommand.MoveSubIndex005 = Position[4] AND
    	E001.Outputs.MotionCommand.MoveSubIndex006 = Position[5] 
    	THEN StepSquareMove := 70 ;
    END_IF;
END_IF;

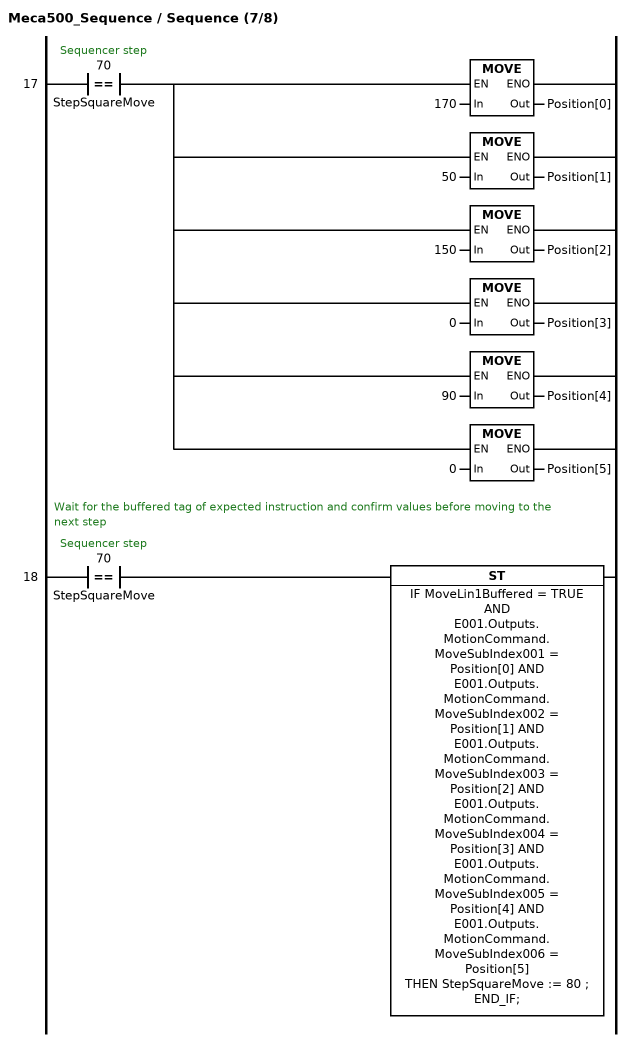
(* Rung 17 *)
IF 70 = StepSquareMove THEN
    Position[0] := 170;
    Position[1] := 50;
    Position[2] := 150;
    Position[3] := 0;
    Position[4] := 90;
    Position[5] := 0;
END_IF;
(* Rung 18: Wait for the buffered tag of expected instruction and confirm values before moving to the next step *)
IF 70 = StepSquareMove THEN
    IF MoveLin1Buffered = TRUE AND
    	E001.Outputs.MotionCommand.MoveSubIndex001 = Position[0] AND
    	E001.Outputs.MotionCommand.MoveSubIndex002 = Position[1] AND
    	E001.Outputs.MotionCommand.MoveSubIndex003 = Position[2] AND
    	E001.Outputs.MotionCommand.MoveSubIndex004 = Position[3] AND
    	E001.Outputs.MotionCommand.MoveSubIndex005 = Position[4] AND
    	E001.Outputs.MotionCommand.MoveSubIndex006 = Position[5] 
    	THEN StepSquareMove := 80 ;
    END_IF;
END_IF;

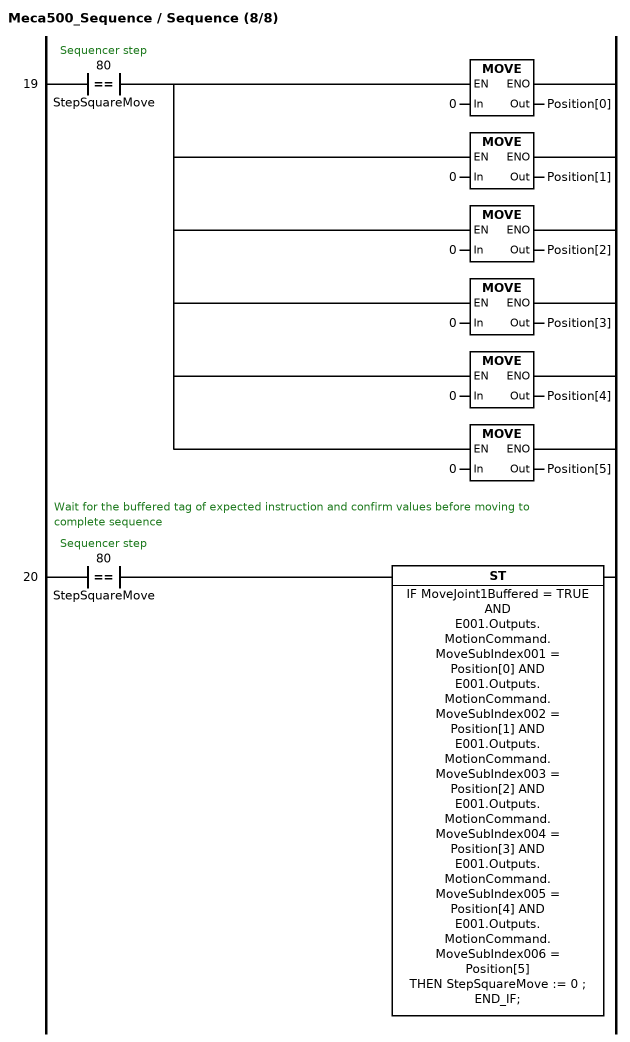
(* Rung 19 *)
IF 80 = StepSquareMove THEN
    Position[0] := 0;
    Position[1] := 0;
    Position[2] := 0;
    Position[3] := 0;
    Position[4] := 0;
    Position[5] := 0;
END_IF;
(* Rung 20: Wait for the buffered tag of expected instruction and confirm values before moving to complete sequence *)
IF 80 = StepSquareMove THEN
    IF MoveJoint1Buffered = TRUE AND
    	E001.Outputs.MotionCommand.MoveSubIndex001 = Position[0] AND
    	E001.Outputs.MotionCommand.MoveSubIndex002 = Position[1] AND
    	E001.Outputs.MotionCommand.MoveSubIndex003 = Position[2] AND
    	E001.Outputs.MotionCommand.MoveSubIndex004 = Position[3] AND
    	E001.Outputs.MotionCommand.MoveSubIndex005 = Position[4] AND
    	E001.Outputs.MotionCommand.MoveSubIndex006 = Position[5] 
    	THEN StepSquareMove := 0 ;
    END_IF;
END_IF;
END_PROGRAM

PROGRAM Meca500_Instructions
VAR
    MoveJoints1 : Meca500_MoveJoints;
    MovePose1 : Meca500_MovePose;
    MoveLin1 : Meca500_MoveLin;
    SetCartLinVel1 : Meca500_SetCartLinVel;
END_VAR
VAR_EXTERNAL
    StepSquareMove : INT;
    E001 : Meca500;
    Position : ARRAY[0..5] OF real;
    MoveJoint1Buffered : BOOL;
    MovePose1Buffered : BOOL;
    MoveLin1Buffered : BOOL;
    SetCartLinVel1Buffered : BOOL;
END_VAR

(* Section Intructions: ladder, written here as Structured Text *)

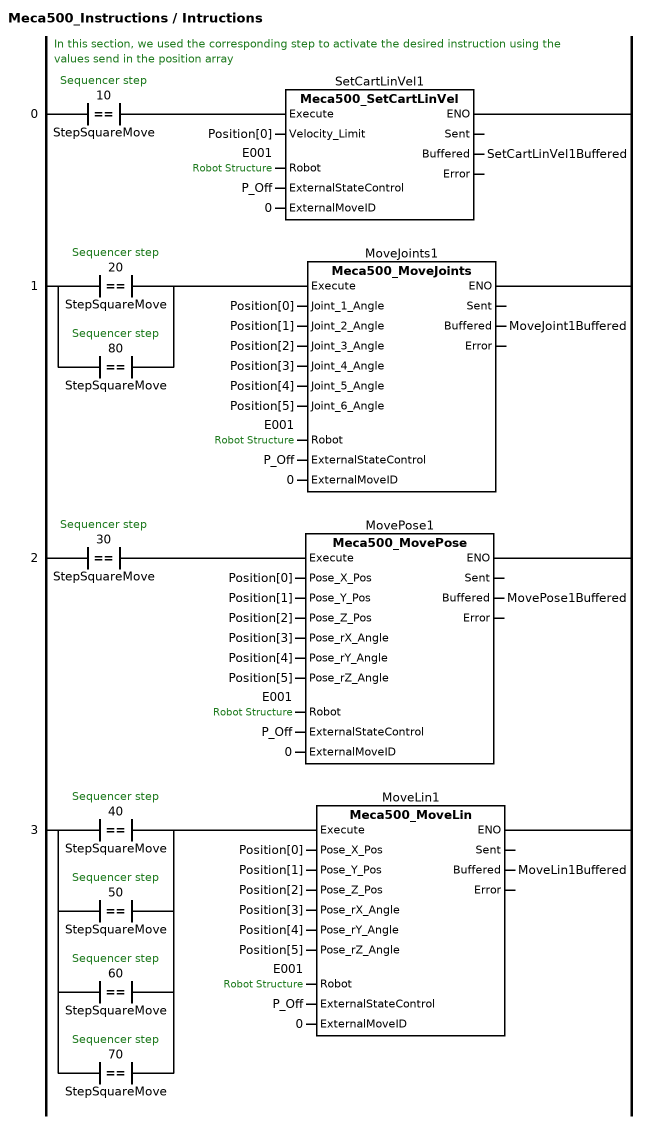
(* Rung 0: In this section, we used the corresponding step to activate the desired instruction using the values send in the position array *)
SetCartLinVel1(Execute := 10 = StepSquareMove, Velocity_Limit := Position[0], Robot := E001, ExternalStateControl := P_Off, ExternalMoveID := 0, Buffered => SetCartLinVel1Buffered);
(* Rung 1 *)
MoveJoints1(Execute := (20 = StepSquareMove) OR (80 = StepSquareMove), Joint_1_Angle := Position[0], Joint_2_Angle := Position[1], Joint_3_Angle := Position[2], Joint_4_Angle := Position[3], Joint_5_Angle := Position[4], Joint_6_Angle := Position[5], Robot := E001, ExternalStateControl := P_Off, ExternalMoveID := 0, Buffered => MoveJoint1Buffered);
(* Rung 2 *)
MovePose1(Execute := 30 = StepSquareMove, Pose_X_Pos := Position[0], Pose_Y_Pos := Position[1], Pose_Z_Pos := Position[2], Pose_rX_Angle := Position[3], Pose_rY_Angle := Position[4], Pose_rZ_Angle := Position[5], Robot := E001, ExternalStateControl := P_Off, ExternalMoveID := 0, Buffered => MovePose1Buffered);
(* Rung 3 *)
MoveLin1(Execute := (40 = StepSquareMove) OR (50 = StepSquareMove) OR (60 = StepSquareMove) OR (70 = StepSquareMove), Pose_X_Pos := Position[0], Pose_Y_Pos := Position[1], Pose_Z_Pos := Position[2], Pose_rX_Angle := Position[3], Pose_rY_Angle := Position[4], Pose_rZ_Angle := Position[5], Robot := E001, ExternalStateControl := P_Off, ExternalMoveID := 0, Buffered => MoveLin1Buffered);
END_PROGRAM

FUNCTION_BLOCK Meca500_Delay
VAR
    Output_Params : array[1..6] of real;
    FirstScan : BOOL := False;
END_VAR
VAR_INPUT
    Execute : BOOL;
    Seconds : REAL;
END_VAR
VAR_OUTPUT
    Sent : BOOL;
    Buffered : BOOL;
    Error : BOOL;
END_VAR
VAR_IN_OUT
    Robot : Meca500;
END_VAR
VAR_INPUT
    ExternalStateControl : BOOL;
    ExternalMoveID : UINT;
END_VAR
IF Execute THEN	
	(*Collect Inputs and store them locally*)
	Output_Params[1]:=Seconds;
	Output_Params[2]:=0;
	Output_Params[3]:=0;
	Output_Params[4]:=0;
	Output_Params[5]:=0;
	Output_Params[6]:=0;


	(* If Values have change, Reinitialise Outputs*)

	IF FirstScan=0 OR 
		Robot.Outputs.MotionCommand.MoveSubIndex001 <> Output_Params[1] OR 
		Robot.Outputs.MotionCommand.MoveSubIndex002 <> Output_Params[2] OR 
		Robot.Outputs.MotionCommand.MoveSubIndex003 <> Output_Params[3] OR
		Robot.Outputs.MotionCommand.MoveSubIndex004 <> Output_Params[4] OR 
		Robot.Outputs.MotionCommand.MoveSubIndex005 <> Output_Params[5] OR 
		Robot.Outputs.MotionCommand.MoveSubIndex006 <> Output_Params[6] 
	THEN
		Buffered := FALSE;
		Sent := FALSE;
	END_IF;


	(*if not in legacy mode, Act Setpoint*)
	IF Robot.Outputs.MotionControl.MoveID <> 0 THEN
	    Robot.Outputs.MotionControl.SetPoint := TRUE;
	END_IF;

	(* To send _Move, send _Move ID *)
	IF NOT Buffered AND NOT Sent THEN
	    
	    Robot.Outputs.MotionCommand.MoveCommand	:= EnumToNum(Meca500Cmd#Delay);
	    Robot.Outputs.MotionCommand.MoveSubIndex001 := Output_Params[1];
		Robot.Outputs.MotionCommand.MoveSubIndex002 := Output_Params[2];
		Robot.Outputs.MotionCommand.MoveSubIndex003 := Output_Params[3];
		Robot.Outputs.MotionCommand.MoveSubIndex004 := Output_Params[4];
		Robot.Outputs.MotionCommand.MoveSubIndex005 := Output_Params[5];
		Robot.Outputs.MotionCommand.MoveSubIndex006 := Output_Params[6];
	    
	    IF ExternalStateControl THEN
	        IF ExternalMoveID <> 0 AND ExternalMoveID <> 32060 AND ExternalMoveID <> 32061 THEN
	            Robot.Outputs.MotionControl.MoveID := ExternalMoveID;
	            Sent := TRUE;
	        END_IF;
	        
	    ELSE (*Not External Control*)
	        IF Robot.Outputs.MotionControl.MoveID = 32060 THEN
	            Robot.Outputs.MotionControl.MoveID := 32061;
	        ELSIF Robot.Outputs.MotionControl.MoveID = 32061 THEN
	            Robot.Outputs.MotionControl.MoveID := 32060;
	        ELSIF Robot.Outputs.MotionControl.MoveID <> 32060 OR Robot.Outputs.MotionControl.MoveID <> 32061 THEN
	            Robot.Outputs.MotionControl.MoveID := 32060;
	        END_IF;
	        Sent := TRUE;
	    END_IF;
	END_IF;

	(* Check if command has been sent, if so, check if it was received *)
	IF Sent AND
	    Robot.Outputs.MotionCommand.MoveCommand = EnumToNum(Meca500Cmd#Delay) AND
	    Robot.Outputs.MotionCommand.MoveSubIndex001 = Output_Params[1] AND 
		Robot.Outputs.MotionCommand.MoveSubIndex002 = Output_Params[2] AND 
		Robot.Outputs.MotionCommand.MoveSubIndex003 = Output_Params[3] AND 
		Robot.Outputs.MotionCommand.MoveSubIndex004 = Output_Params[4] AND 
		Robot.Outputs.MotionCommand.MoveSubIndex005 = Output_Params[5] AND 
		Robot.Outputs.MotionCommand.MoveSubIndex006 = Output_Params[6] AND
		Robot.Inputs.Motion.MoveID = Robot.Outputs.MotionControl.MoveID 
	THEN
		 Buffered := TRUE;
	END_IF;


	(*If External _Move ID is equal to Internal, raise an error*)
	IF ExternalMoveID = 32060 OR ExternalMoveID = 32061 THEN
	    Error := TRUE;
	END_IF;

	FirstScan := TRUE;
ELSE
	FirstScan := False;
	Sent := FALSE;
	Buffered := FALSE;
END_IF;
END_FUNCTION_BLOCK

FUNCTION_BLOCK Meca500_Gripper
VAR
    Output_Params : array[1..6] of real;
    FirstScan : BOOL := False;
END_VAR
VAR_INPUT
    Execute : BOOL;
    Open : REAL;
END_VAR
VAR_OUTPUT
    Sent : BOOL;
    Buffered : BOOL;
    Error : BOOL;
END_VAR
VAR_IN_OUT
    Robot : Meca500;
END_VAR
VAR_INPUT
    ExternalStateControl : BOOL;
    ExternalMoveID : UINT;
END_VAR
IF Execute THEN	
	(*Collect Inputs and store them locally*)
	Output_Params[1]:=Open;
	Output_Params[2]:=0;
	Output_Params[3]:=0;
	Output_Params[4]:=0;
	Output_Params[5]:=0;
	Output_Params[6]:=0;


	(* If Values have change, Reinitialise Outputs*)

	IF FirstScan=0 OR 
		Robot.Outputs.MotionCommand.MoveSubIndex001 <> Output_Params[1] OR 
		Robot.Outputs.MotionCommand.MoveSubIndex002 <> Output_Params[2] OR 
		Robot.Outputs.MotionCommand.MoveSubIndex003 <> Output_Params[3] OR
		Robot.Outputs.MotionCommand.MoveSubIndex004 <> Output_Params[4] OR 
		Robot.Outputs.MotionCommand.MoveSubIndex005 <> Output_Params[5] OR 
		Robot.Outputs.MotionCommand.MoveSubIndex006 <> Output_Params[6] 
	THEN
		Buffered := FALSE;
		Sent := FALSE;
	END_IF;


	(*if not in legacy mode, Act Setpoint*)
	IF Robot.Outputs.MotionControl.MoveID <> 0 THEN
	    Robot.Outputs.MotionControl.SetPoint := TRUE;
	END_IF;

	(* To send _Move, send _Move ID *)
	IF NOT Buffered AND NOT Sent THEN
	    
	    Robot.Outputs.MotionCommand.MoveCommand	:= EnumToNum(Meca500Cmd#Gripper);
	    Robot.Outputs.MotionCommand.MoveSubIndex001 := Output_Params[1];
		Robot.Outputs.MotionCommand.MoveSubIndex002 := Output_Params[2];
		Robot.Outputs.MotionCommand.MoveSubIndex003 := Output_Params[3];
		Robot.Outputs.MotionCommand.MoveSubIndex004 := Output_Params[4];
		Robot.Outputs.MotionCommand.MoveSubIndex005 := Output_Params[5];
		Robot.Outputs.MotionCommand.MoveSubIndex006 := Output_Params[6];
	    
	    IF ExternalStateControl THEN
	        IF ExternalMoveID <> 0 AND ExternalMoveID <> 32180 AND ExternalMoveID <> 32181 THEN
	            Robot.Outputs.MotionControl.MoveID := ExternalMoveID;
	            Sent := TRUE;
	        END_IF;
	        
	    ELSE (*Not External Control*)
	        IF Robot.Outputs.MotionControl.MoveID = 32180 THEN
	            Robot.Outputs.MotionControl.MoveID := 32181;
	        ELSIF Robot.Outputs.MotionControl.MoveID = 32181 THEN
	            Robot.Outputs.MotionControl.MoveID := 32180;
	        ELSIF Robot.Outputs.MotionControl.MoveID <> 32180 OR Robot.Outputs.MotionControl.MoveID <> 32181 THEN
	            Robot.Outputs.MotionControl.MoveID := 32180;
	        END_IF;
	        Sent := TRUE;
	    END_IF;
	END_IF;

	(* Check if command has been sent, if so, check if it was received *)
	IF Sent AND
	    Robot.Outputs.MotionCommand.MoveCommand = EnumToNum(Meca500Cmd#Gripper) AND
	    Robot.Outputs.MotionCommand.MoveSubIndex001 = Output_Params[1] AND 
		Robot.Outputs.MotionCommand.MoveSubIndex002 = Output_Params[2] AND 
		Robot.Outputs.MotionCommand.MoveSubIndex003 = Output_Params[3] AND 
		Robot.Outputs.MotionCommand.MoveSubIndex004 = Output_Params[4] AND 
		Robot.Outputs.MotionCommand.MoveSubIndex005 = Output_Params[5] AND 
		Robot.Outputs.MotionCommand.MoveSubIndex006 = Output_Params[6] AND
		Robot.Inputs.Motion.MoveID = Robot.Outputs.MotionControl.MoveID 
	THEN
		 Buffered := TRUE;
	END_IF;


	(*If External _Move ID is equal to Internal, raise an error*)
	IF ExternalMoveID = 32180 OR ExternalMoveID = 32181 THEN
	    Error := TRUE;
	END_IF;

	FirstScan := TRUE;
ELSE
	FirstScan := False;
	Sent := FALSE;
	Buffered := FALSE;
END_IF;
END_FUNCTION_BLOCK

FUNCTION_BLOCK Meca500_MoveGripper
VAR
    Output_Params : array[1..6] of real;
    FirstScan : BOOL := False;
END_VAR
VAR_INPUT
    Execute : BOOL;
    mm : REAL;
END_VAR
VAR_OUTPUT
    Sent : BOOL;
    Buffered : BOOL;
    Error : BOOL;
END_VAR
VAR_IN_OUT
    Robot : Meca500;
END_VAR
VAR_INPUT
    ExternalStateControl : BOOL;
    ExternalMoveID : UINT;
END_VAR
IF Execute THEN	
	(*Collect Inputs and store them locally*)
	Output_Params[1]:=mm;
	Output_Params[2]:=0;
	Output_Params[3]:=0;
	Output_Params[4]:=0;
	Output_Params[5]:=0;
	Output_Params[6]:=0;


	(* If Values have change, Reinitialise Outputs*)

	IF FirstScan=0 OR 
		Robot.Outputs.MotionCommand.MoveSubIndex001 <> Output_Params[1] OR 
		Robot.Outputs.MotionCommand.MoveSubIndex002 <> Output_Params[2] OR 
		Robot.Outputs.MotionCommand.MoveSubIndex003 <> Output_Params[3] OR
		Robot.Outputs.MotionCommand.MoveSubIndex004 <> Output_Params[4] OR 
		Robot.Outputs.MotionCommand.MoveSubIndex005 <> Output_Params[5] OR 
		Robot.Outputs.MotionCommand.MoveSubIndex006 <> Output_Params[6] 
	THEN
		Buffered := FALSE;
		Sent := FALSE;
	END_IF;


	(*if not in legacy mode, Act Setpoint*)
	IF Robot.Outputs.MotionControl.MoveID <> 0 THEN
	    Robot.Outputs.MotionControl.SetPoint := TRUE;
	END_IF;

	(* To send _Move, send _Move ID *)
	IF NOT Buffered AND NOT Sent THEN
	    
	    Robot.Outputs.MotionCommand.MoveCommand	:= EnumToNum(Meca500Cmd#MoveGripper);
	    Robot.Outputs.MotionCommand.MoveSubIndex001 := Output_Params[1];
		Robot.Outputs.MotionCommand.MoveSubIndex002 := Output_Params[2];
		Robot.Outputs.MotionCommand.MoveSubIndex003 := Output_Params[3];
		Robot.Outputs.MotionCommand.MoveSubIndex004 := Output_Params[4];
		Robot.Outputs.MotionCommand.MoveSubIndex005 := Output_Params[5];
		Robot.Outputs.MotionCommand.MoveSubIndex006 := Output_Params[6];
	    
	    IF ExternalStateControl THEN
	        IF ExternalMoveID <> 0 AND ExternalMoveID <> 32320 AND ExternalMoveID <> 32321 THEN
	            Robot.Outputs.MotionControl.MoveID := ExternalMoveID;
	            Sent := TRUE;
	        END_IF;
	        
	    ELSE (*Not External Control*)
	        IF Robot.Outputs.MotionControl.MoveID = 32320 THEN
	            Robot.Outputs.MotionControl.MoveID := 32321;
	        ELSIF Robot.Outputs.MotionControl.MoveID = 32321 THEN
	            Robot.Outputs.MotionControl.MoveID := 32320;
	        ELSIF Robot.Outputs.MotionControl.MoveID <> 32320 OR Robot.Outputs.MotionControl.MoveID <> 32321 THEN
	            Robot.Outputs.MotionControl.MoveID := 32320;
	        END_IF;
	        Sent := TRUE;
	    END_IF;
	END_IF;

	(* Check if command has been sent, if so, check if it was received *)
	IF Sent AND
	    Robot.Outputs.MotionCommand.MoveCommand = EnumToNum(Meca500Cmd#MoveGripper) AND
	    Robot.Outputs.MotionCommand.MoveSubIndex001 = Output_Params[1] AND 
		Robot.Outputs.MotionCommand.MoveSubIndex002 = Output_Params[2] AND 
		Robot.Outputs.MotionCommand.MoveSubIndex003 = Output_Params[3] AND 
		Robot.Outputs.MotionCommand.MoveSubIndex004 = Output_Params[4] AND 
		Robot.Outputs.MotionCommand.MoveSubIndex005 = Output_Params[5] AND 
		Robot.Outputs.MotionCommand.MoveSubIndex006 = Output_Params[6] AND
		Robot.Inputs.Motion.MoveID = Robot.Outputs.MotionControl.MoveID 
	THEN
		 Buffered := TRUE;
	END_IF;


	(*If External _Move ID is equal to Internal, raise an error*)
	IF ExternalMoveID = 32320 OR ExternalMoveID = 32321 THEN
	    Error := TRUE;
	END_IF;

	FirstScan := TRUE;
ELSE
	FirstScan := False;
	Sent := FALSE;
	Buffered := FALSE;
END_IF;
END_FUNCTION_BLOCK

FUNCTION_BLOCK Meca500_MoveJoints
VAR
    Output_Params : array[1..6] of real;
    FirstScan : BOOL := False;
END_VAR
VAR_INPUT
    Execute : BOOL;
    Joint_1_Angle : REAL;
    Joint_2_Angle : REAL;
    Joint_3_Angle : REAL;
    Joint_4_Angle : REAL;
    Joint_5_Angle : REAL;
    Joint_6_Angle : REAL;
END_VAR
VAR_OUTPUT
    Sent : BOOL;
    Buffered : BOOL;
    Error : BOOL;
END_VAR
VAR_IN_OUT
    Robot : Meca500;
END_VAR
VAR_INPUT
    ExternalStateControl : BOOL;
    ExternalMoveID : UINT;
END_VAR
IF Execute THEN	
	(*Collect Inputs and store them locally*)
	Output_Params[1]:=Joint_1_Angle;
	Output_Params[2]:=Joint_2_Angle;
	Output_Params[3]:=Joint_3_Angle;
	Output_Params[4]:=Joint_4_Angle;
	Output_Params[5]:=Joint_5_Angle;
	Output_Params[6]:=Joint_6_Angle;


	(* If Values have change, Reinitialise Outputs*)

	IF FirstScan=0 OR 
		Robot.Outputs.MotionCommand.MoveSubIndex001 <> Output_Params[1] OR 
		Robot.Outputs.MotionCommand.MoveSubIndex002 <> Output_Params[2] OR 
		Robot.Outputs.MotionCommand.MoveSubIndex003 <> Output_Params[3] OR
		Robot.Outputs.MotionCommand.MoveSubIndex004 <> Output_Params[4] OR 
		Robot.Outputs.MotionCommand.MoveSubIndex005 <> Output_Params[5] OR 
		Robot.Outputs.MotionCommand.MoveSubIndex006 <> Output_Params[6] 
	THEN
		Buffered := FALSE;
		Sent := FALSE;
	END_IF;


	(*if not in legacy mode, Act Setpoint*)
	IF Robot.Outputs.MotionControl.MoveID <> 0 THEN
	    Robot.Outputs.MotionControl.SetPoint := TRUE;
	END_IF;

	(* To send _Move, send _Move ID *)
	IF NOT Buffered AND NOT Sent THEN
	    
	    Robot.Outputs.MotionCommand.MoveCommand	:= EnumToNum(Meca500Cmd#MoveJoints);
	    Robot.Outputs.MotionCommand.MoveSubIndex001 := Output_Params[1];
		Robot.Outputs.MotionCommand.MoveSubIndex002 := Output_Params[2];
		Robot.Outputs.MotionCommand.MoveSubIndex003 := Output_Params[3];
		Robot.Outputs.MotionCommand.MoveSubIndex004 := Output_Params[4];
		Robot.Outputs.MotionCommand.MoveSubIndex005 := Output_Params[5];
		Robot.Outputs.MotionCommand.MoveSubIndex006 := Output_Params[6];
	    
	    IF ExternalStateControl THEN
	        IF ExternalMoveID <> 0 AND ExternalMoveID <> 32010 AND ExternalMoveID <> 32011 THEN
	            Robot.Outputs.MotionControl.MoveID := ExternalMoveID;
	            Sent := TRUE;
	        END_IF;
	        
	    ELSE (*Not External Control*)
	        IF Robot.Outputs.MotionControl.MoveID = 32010 THEN
	            Robot.Outputs.MotionControl.MoveID := 32011;
	        ELSIF Robot.Outputs.MotionControl.MoveID = 32011 THEN
	            Robot.Outputs.MotionControl.MoveID := 32010;
	        ELSIF Robot.Outputs.MotionControl.MoveID <> 32010 OR Robot.Outputs.MotionControl.MoveID <> 32011 THEN
	            Robot.Outputs.MotionControl.MoveID := 32010;
	        END_IF;
	        Sent := TRUE;
	    END_IF;
	END_IF;

	(* Check if command has been sent, if so, check if it was received *)
	IF Sent AND
	    Robot.Outputs.MotionCommand.MoveCommand = EnumToNum(Meca500Cmd#MoveJoints) AND
	    Robot.Outputs.MotionCommand.MoveSubIndex001 = Output_Params[1] AND 
		Robot.Outputs.MotionCommand.MoveSubIndex002 = Output_Params[2] AND 
		Robot.Outputs.MotionCommand.MoveSubIndex003 = Output_Params[3] AND 
		Robot.Outputs.MotionCommand.MoveSubIndex004 = Output_Params[4] AND 
		Robot.Outputs.MotionCommand.MoveSubIndex005 = Output_Params[5] AND 
		Robot.Outputs.MotionCommand.MoveSubIndex006 = Output_Params[6] AND
		Robot.Inputs.Motion.MoveID = Robot.Outputs.MotionControl.MoveID 
	THEN
		 Buffered := TRUE;
	END_IF;


	(*If External _Move ID is equal to Internal, raise an error*)
	IF ExternalMoveID = 32010 OR ExternalMoveID = 32011 THEN
	    Error := TRUE;
	END_IF;

	FirstScan := TRUE;
ELSE
	FirstScan := False;
	Sent := FALSE;
	Buffered := FALSE;
END_IF;
END_FUNCTION_BLOCK

FUNCTION_BLOCK Meca500_MoveJointsRel
VAR
    Output_Params : array[1..6] of real;
    FirstScan : BOOL := False;
END_VAR
VAR_INPUT
    Execute : BOOL;
    Joint_1_Angle : REAL;
    Joint_2_Angle : REAL;
    Joint_3_Angle : REAL;
    Joint_4_Angle : REAL;
    Joint_5_Angle : REAL;
    Joint_6_Angle : REAL;
END_VAR
VAR_OUTPUT
    Sent : BOOL;
    Buffered : BOOL;
    Error : BOOL;
END_VAR
VAR_IN_OUT
    Robot : Meca500;
END_VAR
VAR_INPUT
    ExternalStateControl : BOOL;
    ExternalMoveID : UINT;
END_VAR
IF Execute THEN	
	(*Collect Inputs and store them locally*)
	Output_Params[1]:=Joint_1_Angle;
	Output_Params[2]:=Joint_2_Angle;
	Output_Params[3]:=Joint_3_Angle;
	Output_Params[4]:=Joint_4_Angle;
	Output_Params[5]:=Joint_5_Angle;
	Output_Params[6]:=Joint_6_Angle;


	(* If Values have change, Reinitialise Outputs*)

	IF FirstScan=0 OR 
		Robot.Outputs.MotionCommand.MoveSubIndex001 <> Output_Params[1] OR 
		Robot.Outputs.MotionCommand.MoveSubIndex002 <> Output_Params[2] OR 
		Robot.Outputs.MotionCommand.MoveSubIndex003 <> Output_Params[3] OR
		Robot.Outputs.MotionCommand.MoveSubIndex004 <> Output_Params[4] OR 
		Robot.Outputs.MotionCommand.MoveSubIndex005 <> Output_Params[5] OR 
		Robot.Outputs.MotionCommand.MoveSubIndex006 <> Output_Params[6] 
	THEN
		Buffered := FALSE;
		Sent := FALSE;
	END_IF;


	(*if not in legacy mode, Act Setpoint*)
	IF Robot.Outputs.MotionControl.MoveID <> 0 THEN
	    Robot.Outputs.MotionControl.SetPoint := TRUE;
	END_IF;

	(* To send _Move, send _Move ID *)
	IF NOT Buffered AND NOT Sent THEN
	    
	    Robot.Outputs.MotionCommand.MoveCommand	:= EnumToNum(Meca500Cmd#MoveJointsRel);
	    Robot.Outputs.MotionCommand.MoveSubIndex001 := Output_Params[1];
		Robot.Outputs.MotionCommand.MoveSubIndex002 := Output_Params[2];
		Robot.Outputs.MotionCommand.MoveSubIndex003 := Output_Params[3];
		Robot.Outputs.MotionCommand.MoveSubIndex004 := Output_Params[4];
		Robot.Outputs.MotionCommand.MoveSubIndex005 := Output_Params[5];
		Robot.Outputs.MotionCommand.MoveSubIndex006 := Output_Params[6];
	    
	    IF ExternalStateControl THEN
	        IF ExternalMoveID <> 0 AND ExternalMoveID <> 32290 AND ExternalMoveID <> 32291 THEN
	            Robot.Outputs.MotionControl.MoveID := ExternalMoveID;
	            Sent := TRUE;
	        END_IF;
	        
	    ELSE (*Not External Control*)
	        IF Robot.Outputs.MotionControl.MoveID = 32290 THEN
	            Robot.Outputs.MotionControl.MoveID := 32291;
	        ELSIF Robot.Outputs.MotionControl.MoveID = 32291 THEN
	            Robot.Outputs.MotionControl.MoveID := 32290;
	        ELSIF Robot.Outputs.MotionControl.MoveID <> 32290 OR Robot.Outputs.MotionControl.MoveID <> 32291 THEN
	            Robot.Outputs.MotionControl.MoveID := 32290;
	        END_IF;
	        Sent := TRUE;
	    END_IF;
	END_IF;

	(* Check if command has been sent, if so, check if it was received *)
	IF Sent AND
	    Robot.Outputs.MotionCommand.MoveCommand = EnumToNum(Meca500Cmd#MoveJointsRel) AND
	    Robot.Outputs.MotionCommand.MoveSubIndex001 = Output_Params[1] AND 
		Robot.Outputs.MotionCommand.MoveSubIndex002 = Output_Params[2] AND 
		Robot.Outputs.MotionCommand.MoveSubIndex003 = Output_Params[3] AND 
		Robot.Outputs.MotionCommand.MoveSubIndex004 = Output_Params[4] AND 
		Robot.Outputs.MotionCommand.MoveSubIndex005 = Output_Params[5] AND 
		Robot.Outputs.MotionCommand.MoveSubIndex006 = Output_Params[6] AND
		Robot.Inputs.Motion.MoveID = Robot.Outputs.MotionControl.MoveID 
	THEN
		 Buffered := TRUE;
	END_IF;


	(*If External _Move ID is equal to Internal, raise an error*)
	IF ExternalMoveID = 32290 OR ExternalMoveID = 32291 THEN
	    Error := TRUE;
	END_IF;

	FirstScan := TRUE;
ELSE
	FirstScan := False;
	Sent := FALSE;
	Buffered := FALSE;
END_IF;
END_FUNCTION_BLOCK

FUNCTION_BLOCK Meca500_MoveJointsVel
VAR
    Output_Params : array[1..6] of real;
    FirstScan : BOOL := False;
END_VAR
VAR_INPUT
    Execute : BOOL;
    Joint_1_Vel : REAL;
    Joint_2_Vel : REAL;
    Joint_3_Vel : REAL;
    Joint_4_Vel : REAL;
    Joint_5_Vel : REAL;
    Joint_6_Vel : REAL;
END_VAR
VAR_OUTPUT
    Sent : BOOL;
    Buffered : BOOL;
    Error : BOOL;
END_VAR
VAR_IN_OUT
    Robot : Meca500;
END_VAR
VAR_INPUT
    ExternalStateControl : BOOL;
    ExternalMoveID : UINT;
END_VAR
IF Execute THEN	
	(*Collect Inputs and store them locally*)
	Output_Params[1]:=Joint_1_Vel;
	Output_Params[2]:=Joint_2_Vel;
	Output_Params[3]:=Joint_3_Vel;
	Output_Params[4]:=Joint_4_Vel;
	Output_Params[5]:=Joint_5_Vel;
	Output_Params[6]:=Joint_6_Vel;


	(* If Values have change, Reinitialise Outputs*)

	IF FirstScan=0 OR 
		Robot.Outputs.MotionCommand.MoveSubIndex001 <> Output_Params[1] OR 
		Robot.Outputs.MotionCommand.MoveSubIndex002 <> Output_Params[2] OR 
		Robot.Outputs.MotionCommand.MoveSubIndex003 <> Output_Params[3] OR
		Robot.Outputs.MotionCommand.MoveSubIndex004 <> Output_Params[4] OR 
		Robot.Outputs.MotionCommand.MoveSubIndex005 <> Output_Params[5] OR 
		Robot.Outputs.MotionCommand.MoveSubIndex006 <> Output_Params[6] 
	THEN
		Buffered := FALSE;
		Sent := FALSE;
	END_IF;


	(*if not in legacy mode, Act Setpoint*)
	IF Robot.Outputs.MotionControl.MoveID <> 0 THEN
	    Robot.Outputs.MotionControl.SetPoint := TRUE;
	END_IF;

	(* To send _Move, send _Move ID *)
	IF NOT Buffered AND NOT Sent THEN
	    
	    Robot.Outputs.MotionCommand.MoveCommand	:= EnumToNum(Meca500Cmd#MoveJointsVel);
	    Robot.Outputs.MotionCommand.MoveSubIndex001 := Output_Params[1];
		Robot.Outputs.MotionCommand.MoveSubIndex002 := Output_Params[2];
		Robot.Outputs.MotionCommand.MoveSubIndex003 := Output_Params[3];
		Robot.Outputs.MotionCommand.MoveSubIndex004 := Output_Params[4];
		Robot.Outputs.MotionCommand.MoveSubIndex005 := Output_Params[5];
		Robot.Outputs.MotionCommand.MoveSubIndex006 := Output_Params[6];
	    
	    IF ExternalStateControl THEN
	        IF ExternalMoveID <> 0 AND ExternalMoveID <> 32210 AND ExternalMoveID <> 32211 THEN
	            Robot.Outputs.MotionControl.MoveID := ExternalMoveID;
	            Sent := TRUE;
	        END_IF;
	        
	    ELSE (*Not External Control*)
	        IF Robot.Outputs.MotionControl.MoveID = 32210 THEN
	            Robot.Outputs.MotionControl.MoveID := 32211;
	        ELSIF Robot.Outputs.MotionControl.MoveID = 32211 THEN
	            Robot.Outputs.MotionControl.MoveID := 32210;
	        ELSIF Robot.Outputs.MotionControl.MoveID <> 32210 OR Robot.Outputs.MotionControl.MoveID <> 32211 THEN
	            Robot.Outputs.MotionControl.MoveID := 32210;
	        END_IF;
	        Sent := TRUE;
	    END_IF;
	END_IF;

	(* Check if command has been sent, if so, check if it was received *)
	IF Sent AND
	    Robot.Outputs.MotionCommand.MoveCommand = EnumToNum(Meca500Cmd#MoveJointsVel) AND
	    Robot.Outputs.MotionCommand.MoveSubIndex001 = Output_Params[1] AND 
		Robot.Outputs.MotionCommand.MoveSubIndex002 = Output_Params[2] AND 
		Robot.Outputs.MotionCommand.MoveSubIndex003 = Output_Params[3] AND 
		Robot.Outputs.MotionCommand.MoveSubIndex004 = Output_Params[4] AND 
		Robot.Outputs.MotionCommand.MoveSubIndex005 = Output_Params[5] AND 
		Robot.Outputs.MotionCommand.MoveSubIndex006 = Output_Params[6] AND
		Robot.Inputs.Motion.MoveID = Robot.Outputs.MotionControl.MoveID 
	THEN
		 Buffered := TRUE;
	END_IF;


	(*If External _Move ID is equal to Internal, raise an error*)
	IF ExternalMoveID = 32210 OR ExternalMoveID = 32211 THEN
	    Error := TRUE;
	END_IF;

	FirstScan := TRUE;
ELSE
	FirstScan := False;
	Sent := FALSE;
	Buffered := FALSE;
END_IF;
END_FUNCTION_BLOCK

FUNCTION_BLOCK Meca500_MoveLin
VAR
    Output_Params : array[1..6] of real;
    FirstScan : BOOL := False;
END_VAR
VAR_INPUT
    Execute : BOOL;
    Pose_X_Pos : REAL;
    Pose_Y_Pos : REAL;
    Pose_Z_Pos : REAL;
    Pose_rX_Angle : REAL;
    Pose_rY_Angle : REAL;
    Pose_rZ_Angle : REAL;
END_VAR
VAR_OUTPUT
    Sent : BOOL;
    Buffered : BOOL;
    Error : BOOL;
END_VAR
VAR_IN_OUT
    Robot : Meca500;
END_VAR
VAR_INPUT
    ExternalStateControl : BOOL;
    ExternalMoveID : UINT;
END_VAR
IF Execute THEN	
	(*Collect Inputs and store them locally*)
	Output_Params[1]:=Pose_X_Pos;
	Output_Params[2]:=Pose_Y_Pos;
	Output_Params[3]:=Pose_Z_Pos;
	Output_Params[4]:=Pose_rX_Angle;
	Output_Params[5]:=Pose_rY_Angle;
	Output_Params[6]:=Pose_rZ_Angle;

	(* If Values have change, Reinitialise Outputs*)

	IF FirstScan=0 OR 
		Robot.Outputs.MotionCommand.MoveSubIndex001 <> Output_Params[1] OR 
		Robot.Outputs.MotionCommand.MoveSubIndex002 <> Output_Params[2] OR 
		Robot.Outputs.MotionCommand.MoveSubIndex003 <> Output_Params[3] OR
		Robot.Outputs.MotionCommand.MoveSubIndex004 <> Output_Params[4] OR 
		Robot.Outputs.MotionCommand.MoveSubIndex005 <> Output_Params[5] OR 
		Robot.Outputs.MotionCommand.MoveSubIndex006 <> Output_Params[6] 
	THEN
		Buffered := FALSE;
		Sent := FALSE;
	END_IF;


	(*if not in legacy mode, Act Setpoint*)
	IF Robot.Outputs.MotionControl.MoveID <> 0 THEN
	    Robot.Outputs.MotionControl.SetPoint := TRUE;
	END_IF;

	(* To send _Move, send _Move ID *)
	IF NOT Buffered AND NOT Sent THEN
	    
	    Robot.Outputs.MotionCommand.MoveCommand	:= EnumToNum(Meca500Cmd#MoveLin);
	    Robot.Outputs.MotionCommand.MoveSubIndex001 := Output_Params[1];
		Robot.Outputs.MotionCommand.MoveSubIndex002 := Output_Params[2];
		Robot.Outputs.MotionCommand.MoveSubIndex003 := Output_Params[3];
		Robot.Outputs.MotionCommand.MoveSubIndex004 := Output_Params[4];
		Robot.Outputs.MotionCommand.MoveSubIndex005 := Output_Params[5];
		Robot.Outputs.MotionCommand.MoveSubIndex006 := Output_Params[6];
	    
	    IF ExternalStateControl THEN
	        IF ExternalMoveID <> 0 AND ExternalMoveID <> 32030 AND ExternalMoveID <> 32031 THEN
	            Robot.Outputs.MotionControl.MoveID := ExternalMoveID;
	            Sent := TRUE;
	        END_IF;
	        
	    ELSE (*Not External Control*)
	        IF Robot.Outputs.MotionControl.MoveID = 32030 THEN
	            Robot.Outputs.MotionControl.MoveID := 32031;
	        ELSIF Robot.Outputs.MotionControl.MoveID = 32031 THEN
	            Robot.Outputs.MotionControl.MoveID := 32030;
	        ELSIF Robot.Outputs.MotionControl.MoveID <> 32030 OR Robot.Outputs.MotionControl.MoveID <> 32031 THEN
	            Robot.Outputs.MotionControl.MoveID := 32030;
	        END_IF;
	        Sent := TRUE;
	    END_IF;
	END_IF;

	(* Check if command has been sent, if so, check if it was received *)
	IF Sent AND
	    Robot.Outputs.MotionCommand.MoveCommand = EnumToNum(Meca500Cmd#MoveLin) AND
	    Robot.Outputs.MotionCommand.MoveSubIndex001 = Output_Params[1] AND 
		Robot.Outputs.MotionCommand.MoveSubIndex002 = Output_Params[2] AND 
		Robot.Outputs.MotionCommand.MoveSubIndex003 = Output_Params[3] AND 
		Robot.Outputs.MotionCommand.MoveSubIndex004 = Output_Params[4] AND 
		Robot.Outputs.MotionCommand.MoveSubIndex005 = Output_Params[5] AND 
		Robot.Outputs.MotionCommand.MoveSubIndex006 = Output_Params[6] AND
		Robot.Inputs.Motion.MoveID = Robot.Outputs.MotionControl.MoveID 
	THEN
		 Buffered := TRUE;
	END_IF;


	(*If External _Move ID is equal to Internal, raise an error*)
	IF ExternalMoveID = 32030 OR ExternalMoveID = 32031 THEN
	    Error := TRUE;
	END_IF;

	FirstScan := TRUE;
ELSE
	FirstScan := False;
	Sent := FALSE;
	Buffered := FALSE;
END_IF;
END_FUNCTION_BLOCK

FUNCTION_BLOCK Meca500_MoveLinRelTRF
VAR
    Output_Params : array[1..6] of real;
    FirstScan : BOOL := False;
END_VAR
VAR_INPUT
    Execute : BOOL;
    Pose_X_Pos : REAL;
    Pose_Y_Pos : REAL;
    Pose_Z_Pos : REAL;
    Pose_rX_Angle : REAL;
    Pose_rY_Angle : REAL;
    Pose_rZ_Angle : REAL;
END_VAR
VAR_OUTPUT
    Sent : BOOL;
    Buffered : BOOL;
    Error : BOOL;
END_VAR
VAR_IN_OUT
    Robot : Meca500;
END_VAR
VAR_INPUT
    ExternalStateControl : BOOL;
    ExternalMoveID : UINT;
END_VAR
IF Execute THEN	
	(*Collect Inputs and store them locally*)
	Output_Params[1]:=Pose_X_Pos;
	Output_Params[2]:=Pose_Y_Pos;
	Output_Params[3]:=Pose_Z_Pos;
	Output_Params[4]:=Pose_rX_Angle;
	Output_Params[5]:=Pose_rY_Angle;
	Output_Params[6]:=Pose_rZ_Angle;

	(* If Values have change, Reinitialise Outputs*)

	IF FirstScan=0 OR 
		Robot.Outputs.MotionCommand.MoveSubIndex001 <> Output_Params[1] OR 
		Robot.Outputs.MotionCommand.MoveSubIndex002 <> Output_Params[2] OR 
		Robot.Outputs.MotionCommand.MoveSubIndex003 <> Output_Params[3] OR
		Robot.Outputs.MotionCommand.MoveSubIndex004 <> Output_Params[4] OR 
		Robot.Outputs.MotionCommand.MoveSubIndex005 <> Output_Params[5] OR 
		Robot.Outputs.MotionCommand.MoveSubIndex006 <> Output_Params[6] 
	THEN
		Buffered := FALSE;
		Sent := FALSE;
	END_IF;


	(*if not in legacy mode, Act Setpoint*)
	IF Robot.Outputs.MotionControl.MoveID <> 0 THEN
	    Robot.Outputs.MotionControl.SetPoint := TRUE;
	END_IF;

	(* To send _Move, send _Move ID *)
	IF NOT Buffered AND NOT Sent THEN
	    
	    Robot.Outputs.MotionCommand.MoveCommand	:= EnumToNum(Meca500Cmd#MoveLinRelTrf);
	    Robot.Outputs.MotionCommand.MoveSubIndex001 := Output_Params[1];
		Robot.Outputs.MotionCommand.MoveSubIndex002 := Output_Params[2];
		Robot.Outputs.MotionCommand.MoveSubIndex003 := Output_Params[3];
		Robot.Outputs.MotionCommand.MoveSubIndex004 := Output_Params[4];
		Robot.Outputs.MotionCommand.MoveSubIndex005 := Output_Params[5];
		Robot.Outputs.MotionCommand.MoveSubIndex006 := Output_Params[6];
	    
	    IF ExternalStateControl THEN
	        IF ExternalMoveID <> 0 AND ExternalMoveID <> 32040 AND ExternalMoveID <> 32041 THEN
	            Robot.Outputs.MotionControl.MoveID := ExternalMoveID;
	            Sent := TRUE;
	        END_IF;
	        
	    ELSE (*Not External Control*)
	        IF Robot.Outputs.MotionControl.MoveID = 32040 THEN
	            Robot.Outputs.MotionControl.MoveID := 32041;
	        ELSIF Robot.Outputs.MotionControl.MoveID = 32041 THEN
	            Robot.Outputs.MotionControl.MoveID := 32040;
	        ELSIF Robot.Outputs.MotionControl.MoveID <> 32040 OR Robot.Outputs.MotionControl.MoveID <> 32041 THEN
	            Robot.Outputs.MotionControl.MoveID := 32040;
	        END_IF;
	        Sent := TRUE;
	    END_IF;
	END_IF;

	(* Check if command has been sent, if so, check if it was received *)
	IF Sent AND
	    Robot.Outputs.MotionCommand.MoveCommand = EnumToNum(Meca500Cmd#MoveLinRelTrf) AND
	    Robot.Outputs.MotionCommand.MoveSubIndex001 = Output_Params[1] AND 
		Robot.Outputs.MotionCommand.MoveSubIndex002 = Output_Params[2] AND 
		Robot.Outputs.MotionCommand.MoveSubIndex003 = Output_Params[3] AND 
		Robot.Outputs.MotionCommand.MoveSubIndex004 = Output_Params[4] AND 
		Robot.Outputs.MotionCommand.MoveSubIndex005 = Output_Params[5] AND 
		Robot.Outputs.MotionCommand.MoveSubIndex006 = Output_Params[6] AND
		Robot.Inputs.Motion.MoveID = Robot.Outputs.MotionControl.MoveID 
	THEN
		 Buffered := TRUE;
	END_IF;


	(*If External _Move ID is equal to Internal, raise an error*)
	IF ExternalMoveID = 32040 OR ExternalMoveID = 32041 THEN
	    Error := TRUE;
	END_IF;

	FirstScan := TRUE;
ELSE
	FirstScan := False;
	Sent := FALSE;
	Buffered := FALSE;
END_IF;
END_FUNCTION_BLOCK

FUNCTION_BLOCK Meca500_MoveLinRelWRF
VAR
    Output_Params : array[1..6] of real;
    FirstScan : BOOL := False;
END_VAR
VAR_INPUT
    Execute : BOOL;
    Pose_X_Pos : REAL;
    Pose_Y_Pos : REAL;
    Pose_Z_Pos : REAL;
    Pose_rX_Angle : REAL;
    Pose_rY_Angle : REAL;
    Pose_rZ_Angle : REAL;
END_VAR
VAR_OUTPUT
    Sent : BOOL;
    Buffered : BOOL;
    Error : BOOL;
END_VAR
VAR_IN_OUT
    Robot : Meca500;
END_VAR
VAR_INPUT
    ExternalStateControl : BOOL;
    ExternalMoveID : UINT;
END_VAR
IF Execute THEN	
	(*Collect Inputs and store them locally*)
	Output_Params[1]:=Pose_X_Pos;
	Output_Params[2]:=Pose_Y_Pos;
	Output_Params[3]:=Pose_Z_Pos;
	Output_Params[4]:=Pose_rX_Angle;
	Output_Params[5]:=Pose_rY_Angle;
	Output_Params[6]:=Pose_rZ_Angle;

	(* If Values have change, Reinitialise Outputs*)

	IF FirstScan=0 OR 
		Robot.Outputs.MotionCommand.MoveSubIndex001 <> Output_Params[1] OR 
		Robot.Outputs.MotionCommand.MoveSubIndex002 <> Output_Params[2] OR 
		Robot.Outputs.MotionCommand.MoveSubIndex003 <> Output_Params[3] OR
		Robot.Outputs.MotionCommand.MoveSubIndex004 <> Output_Params[4] OR 
		Robot.Outputs.MotionCommand.MoveSubIndex005 <> Output_Params[5] OR 
		Robot.Outputs.MotionCommand.MoveSubIndex006 <> Output_Params[6] 
	THEN
		Buffered := FALSE;
		Sent := FALSE;
	END_IF;


	(*if not in legacy mode, Act Setpoint*)
	IF Robot.Outputs.MotionControl.MoveID <> 0 THEN
	    Robot.Outputs.MotionControl.SetPoint := TRUE;
	END_IF;

	(* To send _Move, send _Move ID *)
	IF NOT Buffered AND NOT Sent THEN
	    
	    Robot.Outputs.MotionCommand.MoveCommand	:= EnumToNum(Meca500Cmd#MoveLinRelWrf);
	    Robot.Outputs.MotionCommand.MoveSubIndex001 := Output_Params[1];
		Robot.Outputs.MotionCommand.MoveSubIndex002 := Output_Params[2];
		Robot.Outputs.MotionCommand.MoveSubIndex003 := Output_Params[3];
		Robot.Outputs.MotionCommand.MoveSubIndex004 := Output_Params[4];
		Robot.Outputs.MotionCommand.MoveSubIndex005 := Output_Params[5];
		Robot.Outputs.MotionCommand.MoveSubIndex006 := Output_Params[6];
	    
	    IF ExternalStateControl THEN
	        IF ExternalMoveID <> 0 AND ExternalMoveID <> 32050 AND ExternalMoveID <> 32051 THEN
	            Robot.Outputs.MotionControl.MoveID := ExternalMoveID;
	            Sent := TRUE;
	        END_IF;
	        
	    ELSE (*Not External Control*)
	        IF Robot.Outputs.MotionControl.MoveID = 32050 THEN
	            Robot.Outputs.MotionControl.MoveID := 32051;
	        ELSIF Robot.Outputs.MotionControl.MoveID = 32051 THEN
	            Robot.Outputs.MotionControl.MoveID := 32050;
	        ELSIF Robot.Outputs.MotionControl.MoveID <> 32050 OR Robot.Outputs.MotionControl.MoveID <> 32051 THEN
	            Robot.Outputs.MotionControl.MoveID := 32050;
	        END_IF;
	        Sent := TRUE;
	    END_IF;
	END_IF;

	(* Check if command has been sent, if so, check if it was received *)
	IF Sent AND
	    Robot.Outputs.MotionCommand.MoveCommand = EnumToNum(Meca500Cmd#MoveLinRelWrf) AND
	    Robot.Outputs.MotionCommand.MoveSubIndex001 = Output_Params[1] AND 
		Robot.Outputs.MotionCommand.MoveSubIndex002 = Output_Params[2] AND 
		Robot.Outputs.MotionCommand.MoveSubIndex003 = Output_Params[3] AND 
		Robot.Outputs.MotionCommand.MoveSubIndex004 = Output_Params[4] AND 
		Robot.Outputs.MotionCommand.MoveSubIndex005 = Output_Params[5] AND 
		Robot.Outputs.MotionCommand.MoveSubIndex006 = Output_Params[6] AND
		Robot.Inputs.Motion.MoveID = Robot.Outputs.MotionControl.MoveID 
	THEN
		 Buffered := TRUE;
	END_IF;


	(*If External _Move ID is equal to Internal, raise an error*)
	IF ExternalMoveID = 32050 OR ExternalMoveID = 32051 THEN
	    Error := TRUE;
	END_IF;

	FirstScan := TRUE;
ELSE
	FirstScan := False;
	Sent := FALSE;
	Buffered := FALSE;
END_IF;
END_FUNCTION_BLOCK

FUNCTION_BLOCK Meca500_MoveLinVelTRF
VAR
    Output_Params : array[1..6] of real;
    FirstScan : BOOL := False;
END_VAR
VAR_INPUT
    Execute : BOOL;
    X_Vel : REAL;
    Y_Vel : REAL;
    Z_Vel : REAL;
    rX_AngleVel : REAL;
    rY_AngleVel : REAL;
    rZ_AngleVel : REAL;
END_VAR
VAR_OUTPUT
    Sent : BOOL;
    Buffered : BOOL;
    Error : BOOL;
END_VAR
VAR_IN_OUT
    Robot : Meca500;
END_VAR
VAR_INPUT
    ExternalStateControl : BOOL;
    ExternalMoveID : UINT;
END_VAR
IF Execute THEN	
	(*Collect Inputs and store them locally*)
	Output_Params[1]:=X_Vel;
	Output_Params[2]:=Y_Vel;
	Output_Params[3]:=Z_Vel;
	Output_Params[4]:=rX_AngleVel;
	Output_Params[5]:=rY_AngleVel;
	Output_Params[6]:=rZ_AngleVel;

	(* If Values have change, Reinitialise Outputs*)

	IF FirstScan=0 OR 
		Robot.Outputs.MotionCommand.MoveSubIndex001 <> Output_Params[1] OR 
		Robot.Outputs.MotionCommand.MoveSubIndex002 <> Output_Params[2] OR 
		Robot.Outputs.MotionCommand.MoveSubIndex003 <> Output_Params[3] OR
		Robot.Outputs.MotionCommand.MoveSubIndex004 <> Output_Params[4] OR 
		Robot.Outputs.MotionCommand.MoveSubIndex005 <> Output_Params[5] OR 
		Robot.Outputs.MotionCommand.MoveSubIndex006 <> Output_Params[6] 
	THEN
		Buffered := FALSE;
		Sent := FALSE;
	END_IF;


	(*if not in legacy mode, Act Setpoint*)
	IF Robot.Outputs.MotionControl.MoveID <> 0 THEN
	    Robot.Outputs.MotionControl.SetPoint := TRUE;
	END_IF;

	(* To send _Move, send _Move ID *)
	IF NOT Buffered AND NOT Sent THEN
	    
	    Robot.Outputs.MotionCommand.MoveCommand	:= EnumToNum(Meca500Cmd#MoveLinVelTrf);
	    Robot.Outputs.MotionCommand.MoveSubIndex001 := Output_Params[1];
		Robot.Outputs.MotionCommand.MoveSubIndex002 := Output_Params[2];
		Robot.Outputs.MotionCommand.MoveSubIndex003 := Output_Params[3];
		Robot.Outputs.MotionCommand.MoveSubIndex004 := Output_Params[4];
		Robot.Outputs.MotionCommand.MoveSubIndex005 := Output_Params[5];
		Robot.Outputs.MotionCommand.MoveSubIndex006 := Output_Params[6];
	    
	    IF ExternalStateControl THEN
	        IF ExternalMoveID <> 0 AND ExternalMoveID <> 32230 AND ExternalMoveID <> 32231 THEN
	            Robot.Outputs.MotionControl.MoveID := ExternalMoveID;
	            Sent := TRUE;
	        END_IF;
	        
	    ELSE (*Not External Control*)
	        IF Robot.Outputs.MotionControl.MoveID = 32230 THEN
	            Robot.Outputs.MotionControl.MoveID := 32231;
	        ELSIF Robot.Outputs.MotionControl.MoveID = 32231 THEN
	            Robot.Outputs.MotionControl.MoveID := 32230;
	        ELSIF Robot.Outputs.MotionControl.MoveID <> 32230 OR Robot.Outputs.MotionControl.MoveID <> 32231 THEN
	            Robot.Outputs.MotionControl.MoveID := 32230;
	        END_IF;
	        Sent := TRUE;
	    END_IF;
	END_IF;

	(* Check if command has been sent, if so, check if it was received *)
	IF Sent AND
	    Robot.Outputs.MotionCommand.MoveCommand = EnumToNum(Meca500Cmd#MoveLinVelTrf) AND
	    Robot.Outputs.MotionCommand.MoveSubIndex001 = Output_Params[1] AND 
		Robot.Outputs.MotionCommand.MoveSubIndex002 = Output_Params[2] AND 
		Robot.Outputs.MotionCommand.MoveSubIndex003 = Output_Params[3] AND 
		Robot.Outputs.MotionCommand.MoveSubIndex004 = Output_Params[4] AND 
		Robot.Outputs.MotionCommand.MoveSubIndex005 = Output_Params[5] AND 
		Robot.Outputs.MotionCommand.MoveSubIndex006 = Output_Params[6] AND
		Robot.Inputs.Motion.MoveID = Robot.Outputs.MotionControl.MoveID 
	THEN
		 Buffered := TRUE;
	END_IF;


	(*If External _Move ID is equal to Internal, raise an error*)
	IF ExternalMoveID = 32230 OR ExternalMoveID = 32231 THEN
	    Error := TRUE;
	END_IF;

	FirstScan := TRUE;
ELSE
	FirstScan := False;
	Sent := FALSE;
	Buffered := FALSE;
END_IF;
END_FUNCTION_BLOCK

FUNCTION_BLOCK Meca500_MoveLinVelWRF
VAR
    Output_Params : array[1..6] of real;
    FirstScan : BOOL := False;
END_VAR
VAR_INPUT
    Execute : BOOL;
    X_Vel : REAL;
    Y_Vel : REAL;
    Z_Vel : REAL;
    rX_AngleVel : REAL;
    rY_AngleVel : REAL;
    rZ_AngleVel : REAL;
END_VAR
VAR_OUTPUT
    Sent : BOOL;
    Buffered : BOOL;
    Error : BOOL;
END_VAR
VAR_IN_OUT
    Robot : Meca500;
END_VAR
VAR_INPUT
    ExternalStateControl : BOOL;
    ExternalMoveID : UINT;
END_VAR
IF Execute THEN	
	(*Collect Inputs and store them locally*)
	Output_Params[1]:=X_Vel;
	Output_Params[2]:=Y_Vel;
	Output_Params[3]:=Z_Vel;
	Output_Params[4]:=rX_AngleVel;
	Output_Params[5]:=rY_AngleVel;
	Output_Params[6]:=rZ_AngleVel;

	(* If Values have change, Reinitialise Outputs*)

	IF FirstScan=0 OR 
		Robot.Outputs.MotionCommand.MoveSubIndex001 <> Output_Params[1] OR 
		Robot.Outputs.MotionCommand.MoveSubIndex002 <> Output_Params[2] OR 
		Robot.Outputs.MotionCommand.MoveSubIndex003 <> Output_Params[3] OR
		Robot.Outputs.MotionCommand.MoveSubIndex004 <> Output_Params[4] OR 
		Robot.Outputs.MotionCommand.MoveSubIndex005 <> Output_Params[5] OR 
		Robot.Outputs.MotionCommand.MoveSubIndex006 <> Output_Params[6] 
	THEN
		Buffered := FALSE;
		Sent := FALSE;
	END_IF;


	(*if not in legacy mode, Act Setpoint*)
	IF Robot.Outputs.MotionControl.MoveID <> 0 THEN
	    Robot.Outputs.MotionControl.SetPoint := TRUE;
	END_IF;

	(* To send _Move, send _Move ID *)
	IF NOT Buffered AND NOT Sent THEN
	    
	    Robot.Outputs.MotionCommand.MoveCommand	:= EnumToNum(Meca500Cmd#MoveLinVelWrf);
	    Robot.Outputs.MotionCommand.MoveSubIndex001 := Output_Params[1];
		Robot.Outputs.MotionCommand.MoveSubIndex002 := Output_Params[2];
		Robot.Outputs.MotionCommand.MoveSubIndex003 := Output_Params[3];
		Robot.Outputs.MotionCommand.MoveSubIndex004 := Output_Params[4];
		Robot.Outputs.MotionCommand.MoveSubIndex005 := Output_Params[5];
		Robot.Outputs.MotionCommand.MoveSubIndex006 := Output_Params[6];
	    
	    IF ExternalStateControl THEN
	        IF ExternalMoveID <> 0 AND ExternalMoveID <> 32220 AND ExternalMoveID <> 32221 THEN
	            Robot.Outputs.MotionControl.MoveID := ExternalMoveID;
	            Sent := TRUE;
	        END_IF;
	        
	    ELSE (*Not External Control*)
	        IF Robot.Outputs.MotionControl.MoveID = 32220 THEN
	            Robot.Outputs.MotionControl.MoveID := 32221;
	        ELSIF Robot.Outputs.MotionControl.MoveID = 32221 THEN
	            Robot.Outputs.MotionControl.MoveID := 32220;
	        ELSIF Robot.Outputs.MotionControl.MoveID <> 32220 OR Robot.Outputs.MotionControl.MoveID <> 32221 THEN
	            Robot.Outputs.MotionControl.MoveID := 32220;
	        END_IF;
	        Sent := TRUE;
	    END_IF;
	END_IF;

	(* Check if command has been sent, if so, check if it was received *)
	IF Sent AND
	    Robot.Outputs.MotionCommand.MoveCommand = EnumToNum(Meca500Cmd#MoveLinVelWrf) AND
	    Robot.Outputs.MotionCommand.MoveSubIndex001 = Output_Params[1] AND 
		Robot.Outputs.MotionCommand.MoveSubIndex002 = Output_Params[2] AND 
		Robot.Outputs.MotionCommand.MoveSubIndex003 = Output_Params[3] AND 
		Robot.Outputs.MotionCommand.MoveSubIndex004 = Output_Params[4] AND 
		Robot.Outputs.MotionCommand.MoveSubIndex005 = Output_Params[5] AND 
		Robot.Outputs.MotionCommand.MoveSubIndex006 = Output_Params[6] AND
		Robot.Inputs.Motion.MoveID = Robot.Outputs.MotionControl.MoveID 
	THEN
		 Buffered := TRUE;
	END_IF;


	(*If External _Move ID is equal to Internal, raise an error*)
	IF ExternalMoveID = 32220 OR ExternalMoveID = 32221 THEN
	    Error := TRUE;
	END_IF;

	FirstScan := TRUE;
ELSE
	FirstScan := False;
	Sent := FALSE;
	Buffered := FALSE;
END_IF;
END_FUNCTION_BLOCK

FUNCTION_BLOCK Meca500_MovePose
VAR
    Output_Params : array[1..6] of real;
    FirstScan : BOOL := False;
END_VAR
VAR_INPUT
    Execute : BOOL;
    Pose_X_Pos : REAL;
    Pose_Y_Pos : REAL;
    Pose_Z_Pos : REAL;
    Pose_rX_Angle : REAL;
    Pose_rY_Angle : REAL;
    Pose_rZ_Angle : REAL;
END_VAR
VAR_OUTPUT
    Sent : BOOL;
    Buffered : BOOL;
    Error : BOOL;
END_VAR
VAR_IN_OUT
    Robot : Meca500;
END_VAR
VAR_INPUT
    ExternalStateControl : BOOL;
    ExternalMoveID : UINT;
END_VAR
IF Execute THEN	
	(*Collect Inputs and store them locally*)
	Output_Params[1]:=Pose_X_Pos;
	Output_Params[2]:=Pose_Y_Pos;
	Output_Params[3]:=Pose_Z_Pos;
	Output_Params[4]:=Pose_rX_Angle;
	Output_Params[5]:=Pose_rY_Angle;
	Output_Params[6]:=Pose_rZ_Angle;

	(* If Values have change, Reinitialise Outputs*)

	IF FirstScan=0 OR 
		Robot.Outputs.MotionCommand.MoveSubIndex001 <> Output_Params[1] OR 
		Robot.Outputs.MotionCommand.MoveSubIndex002 <> Output_Params[2] OR 
		Robot.Outputs.MotionCommand.MoveSubIndex003 <> Output_Params[3] OR
		Robot.Outputs.MotionCommand.MoveSubIndex004 <> Output_Params[4] OR 
		Robot.Outputs.MotionCommand.MoveSubIndex005 <> Output_Params[5] OR 
		Robot.Outputs.MotionCommand.MoveSubIndex006 <> Output_Params[6] 
	THEN
		Buffered := FALSE;
		Sent := FALSE;
	END_IF;


	(*if not in legacy mode, Act Setpoint*)
	IF Robot.Outputs.MotionControl.MoveID <> 0 THEN
	    Robot.Outputs.MotionControl.SetPoint := TRUE;
	END_IF;

	(* To send _Move, send _Move ID *)
	IF NOT Buffered AND NOT Sent THEN
	    
	    Robot.Outputs.MotionCommand.MoveCommand	:= EnumToNum(Meca500Cmd#MovePose);
	    Robot.Outputs.MotionCommand.MoveSubIndex001 := Output_Params[1];
		Robot.Outputs.MotionCommand.MoveSubIndex002 := Output_Params[2];
		Robot.Outputs.MotionCommand.MoveSubIndex003 := Output_Params[3];
		Robot.Outputs.MotionCommand.MoveSubIndex004 := Output_Params[4];
		Robot.Outputs.MotionCommand.MoveSubIndex005 := Output_Params[5];
		Robot.Outputs.MotionCommand.MoveSubIndex006 := Output_Params[6];
	    
	    IF ExternalStateControl THEN
	        IF ExternalMoveID <> 0 AND ExternalMoveID <> 32020 AND ExternalMoveID <> 32021 THEN
	            Robot.Outputs.MotionControl.MoveID := ExternalMoveID;
	            Sent := TRUE;
	        END_IF;
	        
	    ELSE (*Not External Control*)
	        IF Robot.Outputs.MotionControl.MoveID = 32020 THEN
	            Robot.Outputs.MotionControl.MoveID := 32021;
	        ELSIF Robot.Outputs.MotionControl.MoveID = 32021 THEN
	            Robot.Outputs.MotionControl.MoveID := 32020;
	        ELSIF Robot.Outputs.MotionControl.MoveID <> 32020 OR Robot.Outputs.MotionControl.MoveID <> 32021 THEN
	            Robot.Outputs.MotionControl.MoveID := 32020;
	        END_IF;
	        Sent := TRUE;
	    END_IF;
	END_IF;

	(* Check if command has been sent, if so, check if it was received *)
	IF Sent AND
	    Robot.Outputs.MotionCommand.MoveCommand = EnumToNum(Meca500Cmd#MovePose) AND
	    Robot.Outputs.MotionCommand.MoveSubIndex001 = Output_Params[1] AND 
		Robot.Outputs.MotionCommand.MoveSubIndex002 = Output_Params[2] AND 
		Robot.Outputs.MotionCommand.MoveSubIndex003 = Output_Params[3] AND 
		Robot.Outputs.MotionCommand.MoveSubIndex004 = Output_Params[4] AND 
		Robot.Outputs.MotionCommand.MoveSubIndex005 = Output_Params[5] AND 
		Robot.Outputs.MotionCommand.MoveSubIndex006 = Output_Params[6] AND
		Robot.Inputs.Motion.MoveID = Robot.Outputs.MotionControl.MoveID 
	THEN
		 Buffered := TRUE;
	END_IF;


	(*If External _Move ID is equal to Internal, raise an error*)
	IF ExternalMoveID = 32020 OR ExternalMoveID = 32021 THEN
	    Error := TRUE;
	END_IF;

	FirstScan := TRUE;
ELSE
	FirstScan := False;
	Sent := FALSE;
	Buffered := FALSE;
END_IF;
END_FUNCTION_BLOCK

FUNCTION_BLOCK Meca500_SetAutoConf
VAR
    Output_Params : array[1..6] of real;
    FirstScan : BOOL := False;
END_VAR
VAR_INPUT
    Execute : BOOL;
    Enable : REAL;
END_VAR
VAR_OUTPUT
    Sent : BOOL;
    Buffered : BOOL;
    Error : BOOL;
END_VAR
VAR_IN_OUT
    Robot : Meca500;
END_VAR
VAR_INPUT
    ExternalStateControl : BOOL;
    ExternalMoveID : UINT;
END_VAR
IF Execute THEN	
	(*Collect Inputs and store them locally*)
	Output_Params[1]:=Enable;
	Output_Params[2]:=0;
	Output_Params[3]:=0;
	Output_Params[4]:=0;
	Output_Params[5]:=0;
	Output_Params[6]:=0;

	(* If Values have change, Reinitialise Outputs*)

	IF FirstScan=0 OR 
		Robot.Outputs.MotionCommand.MoveSubIndex001 <> Output_Params[1] OR 
		Robot.Outputs.MotionCommand.MoveSubIndex002 <> Output_Params[2] OR 
		Robot.Outputs.MotionCommand.MoveSubIndex003 <> Output_Params[3] OR
		Robot.Outputs.MotionCommand.MoveSubIndex004 <> Output_Params[4] OR 
		Robot.Outputs.MotionCommand.MoveSubIndex005 <> Output_Params[5] OR 
		Robot.Outputs.MotionCommand.MoveSubIndex006 <> Output_Params[6] 
	THEN
		Buffered := FALSE;
		Sent := FALSE;
	END_IF;


	(*if not in legacy mode, Act Setpoint*)
	IF Robot.Outputs.MotionControl.MoveID <> 0 THEN
	    Robot.Outputs.MotionControl.SetPoint := TRUE;
	END_IF;

	(* To send _Move, send _Move ID *)
	IF NOT Buffered AND NOT Sent THEN
	    
	    Robot.Outputs.MotionCommand.MoveCommand	:= EnumToNum(Meca500Cmd#SetAutoConf);
	    Robot.Outputs.MotionCommand.MoveSubIndex001 := Output_Params[1];
		Robot.Outputs.MotionCommand.MoveSubIndex002 := Output_Params[2];
		Robot.Outputs.MotionCommand.MoveSubIndex003 := Output_Params[3];
		Robot.Outputs.MotionCommand.MoveSubIndex004 := Output_Params[4];
		Robot.Outputs.MotionCommand.MoveSubIndex005 := Output_Params[5];
		Robot.Outputs.MotionCommand.MoveSubIndex006 := Output_Params[6];
	    
	    IF ExternalStateControl THEN
	        IF ExternalMoveID <> 0 AND ExternalMoveID <> 32160 AND ExternalMoveID <> 32161 THEN
	            Robot.Outputs.MotionControl.MoveID := ExternalMoveID;
	            Sent := TRUE;
	        END_IF;
	        
	    ELSE (*Not External Control*)
	        IF Robot.Outputs.MotionControl.MoveID = 32160 THEN
	            Robot.Outputs.MotionControl.MoveID := 32161;
	        ELSIF Robot.Outputs.MotionControl.MoveID = 32161 THEN
	            Robot.Outputs.MotionControl.MoveID := 32160;
	        ELSIF Robot.Outputs.MotionControl.MoveID <> 32160 OR Robot.Outputs.MotionControl.MoveID <> 32161 THEN
	            Robot.Outputs.MotionControl.MoveID := 32160;
	        END_IF;
	        Sent := TRUE;
	    END_IF;
	END_IF;

	(* Check if command has been sent, if so, check if it was received *)
	IF Sent AND
	    Robot.Outputs.MotionCommand.MoveCommand = EnumToNum(Meca500Cmd#SetAutoConf) AND
	    Robot.Outputs.MotionCommand.MoveSubIndex001 = Output_Params[1] AND 
		Robot.Outputs.MotionCommand.MoveSubIndex002 = Output_Params[2] AND 
		Robot.Outputs.MotionCommand.MoveSubIndex003 = Output_Params[3] AND 
		Robot.Outputs.MotionCommand.MoveSubIndex004 = Output_Params[4] AND 
		Robot.Outputs.MotionCommand.MoveSubIndex005 = Output_Params[5] AND 
		Robot.Outputs.MotionCommand.MoveSubIndex006 = Output_Params[6] AND
		Robot.Inputs.Motion.MoveID = Robot.Outputs.MotionControl.MoveID 
	THEN
		 Buffered := TRUE;
	END_IF;


	(*If External _Move ID is equal to Internal, raise an error*)
	IF ExternalMoveID = 32160 OR ExternalMoveID = 32161 THEN
	    Error := TRUE;
	END_IF;

	FirstScan := TRUE;
ELSE
	FirstScan := False;
	Sent := FALSE;
	Buffered := FALSE;
END_IF;
END_FUNCTION_BLOCK

FUNCTION_BLOCK Meca500_SetAutoConfTurn
VAR
    Output_Params : array[1..6] of real;
    FirstScan : BOOL := False;
END_VAR
VAR_INPUT
    Execute : BOOL;
    Enable : REAL;
END_VAR
VAR_OUTPUT
    Sent : BOOL;
    Buffered : BOOL;
    Error : BOOL;
END_VAR
VAR_IN_OUT
    Robot : Meca500;
END_VAR
VAR_INPUT
    ExternalStateControl : BOOL;
    ExternalMoveID : UINT;
END_VAR
IF Execute THEN	
	(*Collect Inputs and store them locally*)
	Output_Params[1]:=Enable;
	Output_Params[2]:=0;
	Output_Params[3]:=0;
	Output_Params[4]:=0;
	Output_Params[5]:=0;
	Output_Params[6]:=0;

	(* If Values have change, Reinitialise Outputs*)

	IF FirstScan=0 OR 
		Robot.Outputs.MotionCommand.MoveSubIndex001 <> Output_Params[1] OR 
		Robot.Outputs.MotionCommand.MoveSubIndex002 <> Output_Params[2] OR 
		Robot.Outputs.MotionCommand.MoveSubIndex003 <> Output_Params[3] OR
		Robot.Outputs.MotionCommand.MoveSubIndex004 <> Output_Params[4] OR 
		Robot.Outputs.MotionCommand.MoveSubIndex005 <> Output_Params[5] OR 
		Robot.Outputs.MotionCommand.MoveSubIndex006 <> Output_Params[6] 
	THEN
		Buffered := FALSE;
		Sent := FALSE;
	END_IF;


	(*if not in legacy mode, Act Setpoint*)
	IF Robot.Outputs.MotionControl.MoveID <> 0 THEN
	    Robot.Outputs.MotionControl.SetPoint := TRUE;
	END_IF;

	(* To send _Move, send _Move ID *)
	IF NOT Buffered AND NOT Sent THEN
	    
	    Robot.Outputs.MotionCommand.MoveCommand	:= EnumToNum(Meca500Cmd#SetAutoConfTurn);
	    Robot.Outputs.MotionCommand.MoveSubIndex001 := Output_Params[1];
		Robot.Outputs.MotionCommand.MoveSubIndex002 := Output_Params[2];
		Robot.Outputs.MotionCommand.MoveSubIndex003 := Output_Params[3];
		Robot.Outputs.MotionCommand.MoveSubIndex004 := Output_Params[4];
		Robot.Outputs.MotionCommand.MoveSubIndex005 := Output_Params[5];
		Robot.Outputs.MotionCommand.MoveSubIndex006 := Output_Params[6];
	    
	    IF ExternalStateControl THEN
	        IF ExternalMoveID <> 0 AND ExternalMoveID <> 32260 AND ExternalMoveID <> 32261 THEN
	            Robot.Outputs.MotionControl.MoveID := ExternalMoveID;
	            Sent := TRUE;
	        END_IF;
	        
	    ELSE (*Not External Control*)
	        IF Robot.Outputs.MotionControl.MoveID = 32260 THEN
	            Robot.Outputs.MotionControl.MoveID := 32261;
	        ELSIF Robot.Outputs.MotionControl.MoveID = 32261 THEN
	            Robot.Outputs.MotionControl.MoveID := 32260;
	        ELSIF Robot.Outputs.MotionControl.MoveID <> 32260 OR Robot.Outputs.MotionControl.MoveID <> 32261 THEN
	            Robot.Outputs.MotionControl.MoveID := 32260;
	        END_IF;
	        Sent := TRUE;
	    END_IF;
	END_IF;

	(* Check if command has been sent, if so, check if it was received *)
	IF Sent AND
	    Robot.Outputs.MotionCommand.MoveCommand = EnumToNum(Meca500Cmd#SetAutoConfTurn) AND
	    Robot.Outputs.MotionCommand.MoveSubIndex001 = Output_Params[1] AND 
		Robot.Outputs.MotionCommand.MoveSubIndex002 = Output_Params[2] AND 
		Robot.Outputs.MotionCommand.MoveSubIndex003 = Output_Params[3] AND 
		Robot.Outputs.MotionCommand.MoveSubIndex004 = Output_Params[4] AND 
		Robot.Outputs.MotionCommand.MoveSubIndex005 = Output_Params[5] AND 
		Robot.Outputs.MotionCommand.MoveSubIndex006 = Output_Params[6] AND
		Robot.Inputs.Motion.MoveID = Robot.Outputs.MotionControl.MoveID 
	THEN
		 Buffered := TRUE;
	END_IF;


	(*If External _Move ID is equal to Internal, raise an error*)
	IF ExternalMoveID = 32260 OR ExternalMoveID = 32261 THEN
	    Error := TRUE;
	END_IF;

	FirstScan := TRUE;
ELSE
	FirstScan := False;
	Sent := FALSE;
	Buffered := FALSE;
END_IF;
END_FUNCTION_BLOCK

FUNCTION_BLOCK Meca500_SetBlending
VAR
    Output_Params : array[1..6] of real;
    FirstScan : BOOL := False;
END_VAR
VAR_INPUT
    Execute : BOOL;
    Blending_Percentage : REAL;
END_VAR
VAR_OUTPUT
    Sent : BOOL;
    Buffered : BOOL;
    Error : BOOL;
END_VAR
VAR_IN_OUT
    Robot : Meca500;
END_VAR
VAR_INPUT
    ExternalStateControl : BOOL;
    ExternalMoveID : UINT;
END_VAR
IF Execute THEN	
	(*Collect Inputs and store them locally*)
	Output_Params[1]:=Blending_Percentage;
	Output_Params[2]:=0;
	Output_Params[3]:=0;
	Output_Params[4]:=0;
	Output_Params[5]:=0;
	Output_Params[6]:=0;

	(* If Values have change, Reinitialise Outputs*)

	IF FirstScan=0 OR 
		Robot.Outputs.MotionCommand.MoveSubIndex001 <> Output_Params[1] OR 
		Robot.Outputs.MotionCommand.MoveSubIndex002 <> Output_Params[2] OR 
		Robot.Outputs.MotionCommand.MoveSubIndex003 <> Output_Params[3] OR
		Robot.Outputs.MotionCommand.MoveSubIndex004 <> Output_Params[4] OR 
		Robot.Outputs.MotionCommand.MoveSubIndex005 <> Output_Params[5] OR 
		Robot.Outputs.MotionCommand.MoveSubIndex006 <> Output_Params[6] 
	THEN
		Buffered := FALSE;
		Sent := FALSE;
	END_IF;


	(*if not in legacy mode, Act Setpoint*)
	IF Robot.Outputs.MotionControl.MoveID <> 0 THEN
	    Robot.Outputs.MotionControl.SetPoint := TRUE;
	END_IF;

	(* To send _Move, send _Move ID *)
	IF NOT Buffered AND NOT Sent THEN
	    
	    Robot.Outputs.MotionCommand.MoveCommand	:= EnumToNum(Meca500Cmd#SetBlending);
	    Robot.Outputs.MotionCommand.MoveSubIndex001 := Output_Params[1];
		Robot.Outputs.MotionCommand.MoveSubIndex002 := Output_Params[2];
		Robot.Outputs.MotionCommand.MoveSubIndex003 := Output_Params[3];
		Robot.Outputs.MotionCommand.MoveSubIndex004 := Output_Params[4];
		Robot.Outputs.MotionCommand.MoveSubIndex005 := Output_Params[5];
		Robot.Outputs.MotionCommand.MoveSubIndex006 := Output_Params[6];
	    
	    IF ExternalStateControl THEN
	        IF ExternalMoveID <> 0 AND ExternalMoveID <> 32070 AND ExternalMoveID <> 32071 THEN
	            Robot.Outputs.MotionControl.MoveID := ExternalMoveID;
	            Sent := TRUE;
	        END_IF;
	        
	    ELSE (*Not External Control*)
	        IF Robot.Outputs.MotionControl.MoveID = 32070 THEN
	            Robot.Outputs.MotionControl.MoveID := 32071;
	        ELSIF Robot.Outputs.MotionControl.MoveID = 32071 THEN
	            Robot.Outputs.MotionControl.MoveID := 32070;
	        ELSIF Robot.Outputs.MotionControl.MoveID <> 32070 OR Robot.Outputs.MotionControl.MoveID <> 32071 THEN
	            Robot.Outputs.MotionControl.MoveID := 32070;
	        END_IF;
	        Sent := TRUE;
	    END_IF;
	END_IF;

	(* Check if command has been sent, if so, check if it was received *)
	IF Sent AND
	    Robot.Outputs.MotionCommand.MoveCommand = EnumToNum(Meca500Cmd#SetBlending) AND
	    Robot.Outputs.MotionCommand.MoveSubIndex001 = Output_Params[1] AND 
		Robot.Outputs.MotionCommand.MoveSubIndex002 = Output_Params[2] AND 
		Robot.Outputs.MotionCommand.MoveSubIndex003 = Output_Params[3] AND 
		Robot.Outputs.MotionCommand.MoveSubIndex004 = Output_Params[4] AND 
		Robot.Outputs.MotionCommand.MoveSubIndex005 = Output_Params[5] AND 
		Robot.Outputs.MotionCommand.MoveSubIndex006 = Output_Params[6] AND
		Robot.Inputs.Motion.MoveID = Robot.Outputs.MotionControl.MoveID 
	THEN
		 Buffered := TRUE;
	END_IF;


	(*If External _Move ID is equal to Internal, raise an error*)
	IF ExternalMoveID = 32070 OR ExternalMoveID = 32071 THEN
	    Error := TRUE;
	END_IF;

	FirstScan := TRUE;
ELSE
	FirstScan := False;
	Sent := FALSE;
	Buffered := FALSE;
END_IF;
END_FUNCTION_BLOCK

FUNCTION_BLOCK Meca500_SetCartAcc
VAR
    Output_Params : array[1..6] of real;
    FirstScan : BOOL := False;
END_VAR
VAR_INPUT
    Execute : BOOL;
    Acceleration_Percentage : REAL;
END_VAR
VAR_OUTPUT
    Sent : BOOL;
    Buffered : BOOL;
    Error : BOOL;
END_VAR
VAR_IN_OUT
    Robot : Meca500;
END_VAR
VAR_INPUT
    ExternalStateControl : BOOL;
    ExternalMoveID : UINT;
END_VAR
IF Execute THEN	
	(*Collect Inputs and store them locally*)
	Output_Params[1]:=Acceleration_Percentage;
	Output_Params[2]:=0;
	Output_Params[3]:=0;
	Output_Params[4]:=0;
	Output_Params[5]:=0;
	Output_Params[6]:=0;

	(* If Values have change, Reinitialise Outputs*)

	IF FirstScan=0 OR 
		Robot.Outputs.MotionCommand.MoveSubIndex001 <> Output_Params[1] OR 
		Robot.Outputs.MotionCommand.MoveSubIndex002 <> Output_Params[2] OR 
		Robot.Outputs.MotionCommand.MoveSubIndex003 <> Output_Params[3] OR
		Robot.Outputs.MotionCommand.MoveSubIndex004 <> Output_Params[4] OR 
		Robot.Outputs.MotionCommand.MoveSubIndex005 <> Output_Params[5] OR 
		Robot.Outputs.MotionCommand.MoveSubIndex006 <> Output_Params[6] 
	THEN
		Buffered := FALSE;
		Sent := FALSE;
	END_IF;


	(*if not in legacy mode, Act Setpoint*)
	IF Robot.Outputs.MotionControl.MoveID <> 0 THEN
	    Robot.Outputs.MotionControl.SetPoint := TRUE;
	END_IF;

	(* To send _Move, send _Move ID *)
	IF NOT Buffered AND NOT Sent THEN
	    
	    Robot.Outputs.MotionCommand.MoveCommand	:= EnumToNum(Meca500Cmd#SetCartAcc);
	    Robot.Outputs.MotionCommand.MoveSubIndex001 := Output_Params[1];
		Robot.Outputs.MotionCommand.MoveSubIndex002 := Output_Params[2];
		Robot.Outputs.MotionCommand.MoveSubIndex003 := Output_Params[3];
		Robot.Outputs.MotionCommand.MoveSubIndex004 := Output_Params[4];
		Robot.Outputs.MotionCommand.MoveSubIndex005 := Output_Params[5];
		Robot.Outputs.MotionCommand.MoveSubIndex006 := Output_Params[6];
	    
	    IF ExternalStateControl THEN
	        IF ExternalMoveID <> 0 AND ExternalMoveID <> 32120 AND ExternalMoveID <> 32121 THEN
	            Robot.Outputs.MotionControl.MoveID := ExternalMoveID;
	            Sent := TRUE;
	        END_IF;
	        
	    ELSE (*Not External Control*)
	        IF Robot.Outputs.MotionControl.MoveID = 32120 THEN
	            Robot.Outputs.MotionControl.MoveID := 32121;
	        ELSIF Robot.Outputs.MotionControl.MoveID = 32121 THEN
	            Robot.Outputs.MotionControl.MoveID := 32120;
	        ELSIF Robot.Outputs.MotionControl.MoveID <> 32120 OR Robot.Outputs.MotionControl.MoveID <> 32121 THEN
	            Robot.Outputs.MotionControl.MoveID := 32120;
	        END_IF;
	        Sent := TRUE;
	    END_IF;
	END_IF;

	(* Check if command has been sent, if so, check if it was received *)
	IF Sent AND
	    Robot.Outputs.MotionCommand.MoveCommand = EnumToNum(Meca500Cmd#SetCartAcc) AND
	    Robot.Outputs.MotionCommand.MoveSubIndex001 = Output_Params[1] AND 
		Robot.Outputs.MotionCommand.MoveSubIndex002 = Output_Params[2] AND 
		Robot.Outputs.MotionCommand.MoveSubIndex003 = Output_Params[3] AND 
		Robot.Outputs.MotionCommand.MoveSubIndex004 = Output_Params[4] AND 
		Robot.Outputs.MotionCommand.MoveSubIndex005 = Output_Params[5] AND 
		Robot.Outputs.MotionCommand.MoveSubIndex006 = Output_Params[6] AND
		Robot.Inputs.Motion.MoveID = Robot.Outputs.MotionControl.MoveID 
	THEN
		 Buffered := TRUE;
	END_IF;


	(*If External _Move ID is equal to Internal, raise an error*)
	IF ExternalMoveID = 32120 OR ExternalMoveID = 32121 THEN
	    Error := TRUE;
	END_IF;

	FirstScan := TRUE;
ELSE
	FirstScan := False;
	Sent := FALSE;
	Buffered := FALSE;
END_IF;
END_FUNCTION_BLOCK

FUNCTION_BLOCK Meca500_SetCartAngVel
VAR
    Output_Params : array[1..6] of real;
    FirstScan : BOOL := False;
END_VAR
VAR_INPUT
    Execute : BOOL;
    Velocity_Limit : REAL;
END_VAR
VAR_OUTPUT
    Sent : BOOL;
    Buffered : BOOL;
    Error : BOOL;
END_VAR
VAR_IN_OUT
    Robot : Meca500;
END_VAR
VAR_INPUT
    ExternalStateControl : BOOL;
    ExternalMoveID : UINT;
END_VAR
IF Execute THEN	
	(*Collect Inputs and store them locally*)
	Output_Params[1]:=Velocity_Limit;
	Output_Params[2]:=0;
	Output_Params[3]:=0;
	Output_Params[4]:=0;
	Output_Params[5]:=0;
	Output_Params[6]:=0;

	(* If Values have change, Reinitialise Outputs*)

	IF FirstScan=0 OR 
		Robot.Outputs.MotionCommand.MoveSubIndex001 <> Output_Params[1] OR 
		Robot.Outputs.MotionCommand.MoveSubIndex002 <> Output_Params[2] OR 
		Robot.Outputs.MotionCommand.MoveSubIndex003 <> Output_Params[3] OR
		Robot.Outputs.MotionCommand.MoveSubIndex004 <> Output_Params[4] OR 
		Robot.Outputs.MotionCommand.MoveSubIndex005 <> Output_Params[5] OR 
		Robot.Outputs.MotionCommand.MoveSubIndex006 <> Output_Params[6] 
	THEN
		Buffered := FALSE;
		Sent := FALSE;
	END_IF;


	(*if not in legacy mode, Act Setpoint*)
	IF Robot.Outputs.MotionControl.MoveID <> 0 THEN
	    Robot.Outputs.MotionControl.SetPoint := TRUE;
	END_IF;

	(* To send _Move, send _Move ID *)
	IF NOT Buffered AND NOT Sent THEN
	    
	    Robot.Outputs.MotionCommand.MoveCommand	:= EnumToNum(Meca500Cmd#SetCartAngVel);
	    Robot.Outputs.MotionCommand.MoveSubIndex001 := Output_Params[1];
		Robot.Outputs.MotionCommand.MoveSubIndex002 := Output_Params[2];
		Robot.Outputs.MotionCommand.MoveSubIndex003 := Output_Params[3];
		Robot.Outputs.MotionCommand.MoveSubIndex004 := Output_Params[4];
		Robot.Outputs.MotionCommand.MoveSubIndex005 := Output_Params[5];
		Robot.Outputs.MotionCommand.MoveSubIndex006 := Output_Params[6];
	    
	    IF ExternalStateControl THEN
	        IF ExternalMoveID <> 0 AND ExternalMoveID <> 32100 AND ExternalMoveID <> 32101 THEN
	            Robot.Outputs.MotionControl.MoveID := ExternalMoveID;
	            Sent := TRUE;
	        END_IF;
	        
